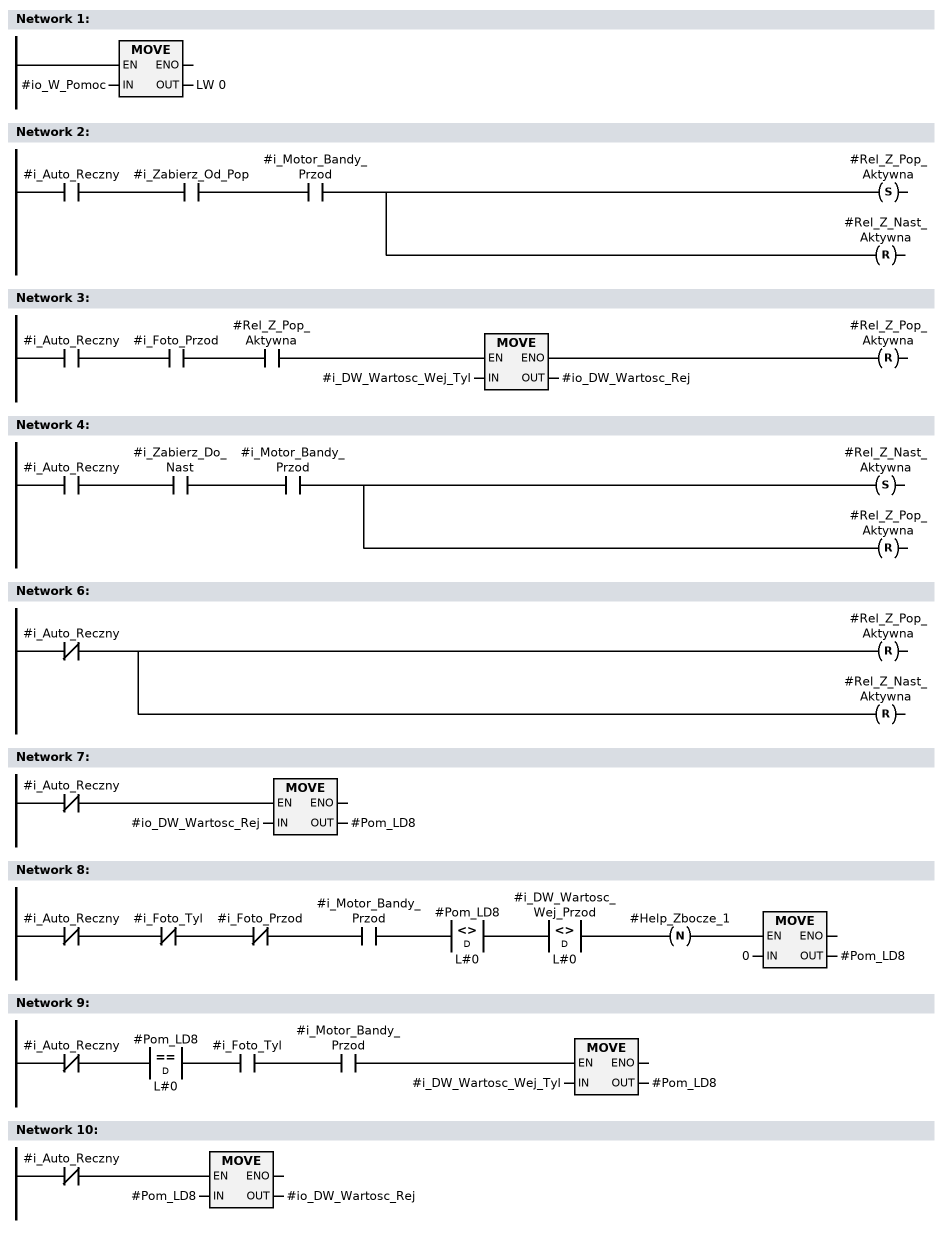
[picture p321: Monitor_Bandy_2 networks 1-10]
NETWORK
TITLE =
//Ten network celowo jest wolny
      L     #io_W_Pomoc;
      T     LW 0;
      NOP   0;
NETWORK
TITLE =
//Tryb Auto
//Pobranie wartosci
//
      A     #i_Auto_Reczny;
      A     #i_Zabierz_Od_Pop;
      A     #i_Motor_Bandy_Przod;
      S     #Rel_Z_Pop_Aktywna;
      R     #Rel_Z_Nast_Aktywna;
NETWORK
TITLE =
//Dojazd do fotokomorki i przepisanie wartosci.Informacja moze byc tez szybciej 
//przekazana (Gender potrzebuje szybciej)
      A     #i_Auto_Reczny;
      A     #i_Foto_Przod;
      A     #Rel_Z_Pop_Aktywna;
      JNB   _001;
      L     #i_DW_Wartosc_Wej_Tyl;
      T     #io_DW_Wartosc_Rej;
      SET;
      SAVE;
      CLR;
_001: A     BR;
      R     #Rel_Z_Pop_Aktywna;
NETWORK
TITLE =
//Relacja z nastepna banda
      A     #i_Auto_Reczny;
      A     #i_Zabierz_Do_Nast;
      A     #i_Motor_Bandy_Przod;
      S     #Rel_Z_Nast_Aktywna;
      R     #Rel_Z_Pop_Aktywna;
NETWORK
TITLE =
//Tryb Reczny
//Warunkiem prawidlowego dzialania trybu reczenego jest pokrycie zawsze co 
//najmniej jednej fotokomorki gdy jest produkt
//
//
NETWORK
TITLE =
//Zresetowanie relacji z automatyki
//
      AN    #i_Auto_Reczny;
      R     #Rel_Z_Pop_Aktywna;
      R     #Rel_Z_Nast_Aktywna;
NETWORK
TITLE =
//Trzeba sobie jakos radzic
      AN    #i_Auto_Reczny;
      JNB   _002;
      L     #io_DW_Wartosc_Rej;
      T     #Pom_LD8;
_002: NOP   0;
NETWORK
TITLE =
//Jazda do przodu na recznym.Bierzaca--->Nastepna
      AN    #i_Auto_Reczny;
      AN    #i_Foto_Tyl;
      AN    #i_Foto_Przod;
      A     #i_Motor_Bandy_Przod;
      A(;
      L     #Pom_LD8;
      L     L#0;
      <>D;
      );
      A(;
      L     #i_DW_Wartosc_Wej_Przod;
      L     L#0;
      <>D;
      );
      FN    #Help_Zbocze_1;
      JNB   _003;
      L     0;
      T     #Pom_LD8;
_003: NOP   0;
NETWORK
TITLE =
//Poprzednia wjezdza na bierzaca w trybie recznym. Poprzednia--->Bierzaca
      AN    #i_Auto_Reczny;
      A(;
      L     #Pom_LD8;
      L     L#0;
      ==D;
      );
      A     #i_Foto_Tyl;
      A     #i_Motor_Bandy_Przod;
      JNB   _004;
      L     #i_DW_Wartosc_Wej_Tyl;
      T     #Pom_LD8;
_004: NOP   0;
NETWORK
TITLE =
//Przepisanie powrotne
      AN    #i_Auto_Reczny;
      JNB   _005;
      L     #Pom_LD8;
      T     #io_DW_Wartosc_Rej;
_005: NOP   0;
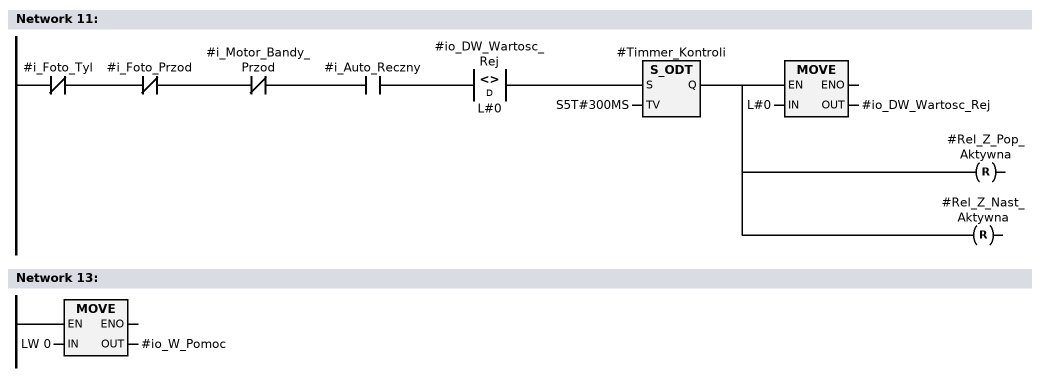
NETWORK
TITLE =
//Sprawdznie wszystkiego
//
      AN    #i_Foto_Tyl;
      AN    #i_Foto_Przod;
      AN    #i_Motor_Bandy_Przod;
      A     #i_Auto_Reczny;
      A(;
      L     #io_DW_Wartosc_Rej;
      L     L#0;
      <>D;
      );
      L     S5T#300MS;
      SD    #Timmer_Kontroli;
      NOP   0;
      NOP   0;
      NOP   0;
      A     #Timmer_Kontroli;
      =     L 12.0;
      A     L 12.0;
      JNB   _006;
      L     L#0;
      T     #io_DW_Wartosc_Rej;
_006: NOP   0;
      A     L 12.0;
      BLD   102;
      R     #Rel_Z_Pop_Aktywna;
      A     L 12.0;
      BLD   102;
      R     #Rel_Z_Nast_Aktywna;
NETWORK
TITLE =
//0.7 - paleta obecna (nieuzywane)
//0.6 - kierunek spedycja (uzywane)
//0.5 - kierunek intro (uzywane)
//0.4 - wiazanie poprzeczne (uzywane)
//0.3 - wiazanie wzdluzne   (uzywane)
//0.2 - deklowanie (uzywane)
//0.1 - foliowanie (uzywane)
//0.0 - paleta obrabiana
//1.7 - rezerwa (nieuzywane)
//1.6 - rezerwa (nieuzywane)
//1.5 - rezerwa (nieuzywane)
//1.3 - rezerwa (nieuzywane)
//1.3 - info bit 3
//1.2 - info bit 2
//1.1 - info bit 1 
//1.0 - info bit 0
//
NETWORK
TITLE =
//Przypisanie wartosci z pamieci podrecznej
//
      L     LW 0;
      T     #io_W_Pomoc;
      NOP   0;
END_FUNCTION

FUNCTION "Monitor_Palety" : VOID	// FC 316
VERSION : 0.1
VAR_INPUT
  Foto_Pozycji_Przod : BOOL ;
  Foto_Pozycji_Tyl : BOOL ;	//Opcjonalna fotokomorka
END_VAR
VAR_IN_OUT
  iod_Wartosc_Rejestru : DINT ;
END_VAR
VAR_TEMP
  Wartosc_Pomocnicz_0 : DINT ;
  Wartosc_Pomocnicz_1 : DINT ;
END_VAR
BEGIN
NETWORK
TITLE =
      L     #iod_Wartosc_Rejestru;
      T     #Wartosc_Pomocnicz_0;
      O     #Foto_Pozycji_Przod;
      O     #Foto_Pozycji_Tyl;
      JCN   et_1;
      SET;
      S     L 0.7;
et_1: NOP   0;
      AN    #Foto_Pozycji_Przod;
      AN    #Foto_Pozycji_Tyl;
      JCN   et_2;
      SET;
      R     L 0.7;
et_2: NOP   0;
      L     #Wartosc_Pomocnicz_0;
      T     #iod_Wartosc_Rejestru;
END_FUNCTION

FUNCTION "Znajdz_Widmo" : VOID	// FC 317
//0.7 - paleta obecna (nieuzywane)
//0.6 - kierunek spedycja (uzywane)
//0.5 - kierunek intro (uzywane)
//0.4 - wiazanie poprzeczne (uzywane)
//0.3 - wiazanie wzdluzne   (uzywane)
//0.2 - deklowanie (uzywane)
//0.1 - foliowanie (uzywane)
//0.0 - paleta obrabiana
//1.7 - rezerwa (nieuzywane)
//1.6 - rezerwa (nieuzywane)
//1.5 - rezerwa (nieuzywane)
//1.3 - rezerwa (nieuzywane)
//1.3 - info bit 3
//1.2 - info bit 2
//1.1 - info bit 1 
//1.0 - info bit 0
VERSION : 0.1
VAR_INPUT
  Paleta_Obecna : BOOL ;
END_VAR
VAR_IN_OUT
  iod_Wartosc_Rejestru : DINT ;
END_VAR
VAR_TEMP
  Wartosc_Pomocnicz_0 : DINT ;
  Wartosc_Pomocnicz_1 : DINT ;
END_VAR
BEGIN
NETWORK
TITLE =
      L     #iod_Wartosc_Rejestru;
      T     #Wartosc_Pomocnicz_0;
      A     #Paleta_Obecna;
      JCN   et_1;
//jesli nie wiadomo co zrobic z paleta i skad 
//jes
      AN    L 0.6;
      AN    L 0.5;
      S     L 0.5;
et_1: NOP   0;
      L     #Wartosc_Pomocnicz_0;
      T     #iod_Wartosc_Rejestru;
END_FUNCTION

FUNCTION "Dekoduj_Maske" : VOID	// FC 320
//0.0 - paleta obecna (nieuzywane)
//0.1 - kierunek spedycja (uzywane)
//0.2 - kierunek intro (uzywane)
//0.3 - wiazanie poprzeczne (uzywane)
//0.4 - wiazanie wzdluzne   (uzywane)
//0.5 - deklowanie (uzywane)
//0.6 - foliowanie (uzywane)
//0.7 - paleta_obrabiana
//1.0 - info bit 0
//1.1 - info bit 1
//1.2 - info bit 2 
//1.3 - info bit 3
//1.4 - rezerwa (nieuzywane)
//1.5 - rezerwa (nieuzywane)
//1.6 - rezerwa (nieuzywane)
//1.7 - rezerwa (nieuzywane)
//
VERSION : 0.1
VAR_INPUT
  Wartosc_Elementu : DINT ;
END_VAR
VAR_OUTPUT
  o_Paleta_Obecna : BOOL ;	//0.7
  o_Kierunek_Spedycja : BOOL ;	//0.6
  o_Kierunek_Intro : BOOL ;	//0.5
  o_Wizanie_Poprzeczne : BOOL ;	//0.4
  o_Wiazanie_Wzdluzne : BOOL ;	//0.3
  o_Deklowanie : BOOL ;	//0.2
  o_Foliowanie : BOOL ;	//0.1
  o_Paleta_Obrabiana : BOOL ;	//0.0
  o_Rezerwa_1_7 : BOOL ;	//1.7
  o_Rezerwa_1_6 : BOOL ;	//1.1
  o_Rezerwa_1_5 : BOOL ;	//1.2
  o_Rezerwa_1_4 : BOOL ;	//1.4
  o_Info_Bit_3 : BOOL ;	//1.3
  o_Info_Bit_2 : BOOL ;	//1.2
  o_Info_Bit_1 : BOOL ;	//1.1
  o_Info_Bit_0 : BOOL ;	//1.0
END_VAR
VAR_TEMP
  Edek_0 : DWORD ;
  Paleta_Obrabiana : BOOL ;	//0.0 - paleta_obrabiana
  Foliowanie : BOOL ;	//0.1
  Deklowanie : BOOL ;	//0.2
  Wiazanie_Wzdluzne : BOOL ;	//0.3
  Wizanie_Poprzeczne : BOOL ;	//0.4
  Kierunek_Intro : BOOL ;	//0.5
  Kierunek_Spedycja : BOOL ;	//0.6
  Paleta_Obecna : BOOL ;	//0.7
  Info_Bit_0 : BOOL ;	//1.0
  Info_Bit_1 : BOOL ;	//1.1
  Info_Bit_2 : BOOL ;	//1.2
  Info_Bit_3 : BOOL ;	//1.3
  Rezerwa_1_4 : BOOL ;	//1.4
  Rezerwa_1_5 : BOOL ;	//1.5
  Rezerwa_1_6 : BOOL ;	//1.6
  Rezerwa_1_7 : BOOL ;	//1.7
END_VAR
BEGIN
NETWORK
TITLE =
//ten network celowo jest wolny
NETWORK
TITLE =
//Zaladowanie maski
      L     #Wartosc_Elementu;
      T     LD 4;
NETWORK
TITLE =
//Wyluskanie zadan
      A     #Paleta_Obrabiana;
      =     #o_Paleta_Obrabiana;
//***
      A     #Foliowanie;
      =     #o_Foliowanie;
//***
      A     #Deklowanie;
      =     #o_Deklowanie;
//***
      A     #Wiazanie_Wzdluzne;
      =     #o_Wiazanie_Wzdluzne;
//***
      A     #Wizanie_Poprzeczne;
      =     #o_Wizanie_Poprzeczne;
//***
      A     #Kierunek_Intro;
      =     #o_Kierunek_Intro;
//***
      A     #Kierunek_Spedycja;
      =     #o_Kierunek_Spedycja;
//***
      A     #Paleta_Obecna;
      =     #o_Paleta_Obecna;
//***
      A     #Info_Bit_0;
      =     #o_Info_Bit_0;
//***
      A     #Info_Bit_1;
      =     #o_Info_Bit_1;
//***
      A     #Info_Bit_2;
      =     #o_Info_Bit_2;
//***
      A     #Info_Bit_3;
      =     #o_Info_Bit_3;
//***
      A     #Rezerwa_1_4;
      =     #o_Rezerwa_1_4;
//***
      A     #Rezerwa_1_5;
      =     #o_Rezerwa_1_5;
//***
      A     #Rezerwa_1_6;
      =     #o_Rezerwa_1_6;
//***
      A     #Rezerwa_1_7;
      =     #o_Rezerwa_1_7;
END_FUNCTION

FUNCTION "Dobor_Elementow_Lini" : VOID	// FC 400
//Funkcja tworzy liste przyciskow bistabilny uzywanych do wyboru trybu pracy w 
//Gender Fedder Line.Dostepne funkcjonalosci wybieramy za pomoca przyciskow
//Spedycja i Intro. Po wyborze przycisku rozwijaja sie funkcjonalnosci.
//
//Spedycja   lub  Intro:
//Spedycja->o_Wiazanie_Pop_Aktywne->o_Deklowanie_Aktywne
//Spedycja->o_Wiazanie_Wzdl_Aktywne
//Spedycja->o_Foliowanie_Aktywne
//
//Intro->o_Instert_Intro_Aktywne
//
//Na koncu funkcji tworzona jest mask sluzaca dalszej obrobce zadan w programie.
//Bity maski:
//
//0.7 - paleta obecna (nieuzywane)
//0.6 - kierunek spedycja (uzywane)
//0.5 - kierunek intro (uzywane)
//0.4 - wiazanie poprzeczne (uzywane)
//0.3 - wiazanie wzdluzne   (uzywane)
//0.2 - deklowanie (uzywane)
//0.1 - foliowanie (uzywane)
//0.0 - paleta obrabiana
//1.7 - rezerwa (nieuzywane)
//1.6 - rezerwa (nieuzywane)
//1.5 - rezerwa (nieuzywane)
//1.3 - rezerwa (nieuzywane)
//1.3 - info bit 3
//1.2 - info bit 2
//1.1 - info bit 1 
//1.0 - info bit 0
//
AUTHOR : Kng
NAME : Help_FC
VERSION : 0.1
VAR_INPUT
  i_Kierunek_Spedycja : BOOL ;
  i_Kierunek_Intro : BOOL ;
  i_Wiazanie_Poprzeczne : BOOL ;
  i_Wiazanie_Wzdluzne : BOOL ;
  i_Deklowanie : BOOL ;
  i_Foliowanie : BOOL ;
  i_Paleta_Obrabiana : BOOL ;	//Informacja czy paleta jest obrabiana
  i_Koder_Bit_0 : BOOL ;
  i_Koder_Bit_1 : BOOL ;
  i_Koder_Bit_2 : BOOL ;
  i_Koder_Bit_3 : BOOL ;
END_VAR
VAR_OUTPUT
  o_Kier_Spedycja_Wyb : BOOL ;
  o_Kier_Intro_Wyb : BOOL ;
  o_Wiazanie_Pop_Wyb : BOOL ;	//To co jest wybrane
  o_Wiazanie_Wzdl_Wyb : BOOL ;
  o_Deklowanie_Wyb : BOOL ;
  o_Foliowanie_Wyb : BOOL ;
  o_Kier_Spedycja_Akt : BOOL ;
  o_Kier_Intro_Akt : BOOL ;
  o_Wiazanie_Pop_Akt : BOOL ;	//To co mozna wybrac
  o_Wiazanie_Wzdl_Akt : BOOL ;
  o_Deklowanie_Akt : BOOL ;
  o_Foliowanie_Akt : BOOL ;
  o_Maska_Zadania : INT ;	//Maska w wynikowa
END_VAR
VAR_IN_OUT
  io_Help_DW : DINT ;	//Slowo pomocnicze
END_VAR
VAR_TEMP
  L_Rezerwa_0_0 : BOOL ;
  L_Rezerwa_0_1 : BOOL ;
  L_Rezerwa_0_2 : BOOL ;
  L_Rezerwa_0_3 : BOOL ;
  L_Rezerwa_0_4 : BOOL ;
  L_Rezerwa_0_5 : BOOL ;
  L_Rezerwa_0_6 : BOOL ;
  L_Rezerwa_0_7 : BOOL ;
  L_Rezerwa_1_0 : BOOL ;
  L_Rezerwa_1_1 : BOOL ;
  L_Rezerwa_1_2 : BOOL ;
  L_Rezerwa_1_3 : BOOL ;
  L_Rezerwa_1_4 : BOOL ;
  L_Rezerwa_1_5 : BOOL ;
  L_Rezerwa_1_6 : BOOL ;
  L_Rezerwa_1_7 : BOOL ;
  L_Rezerwa_Int_2_0 : INT ;
  io_L_Kier_Spedycja : BOOL ;
  io_L_Wiazanie_Poprzeczne : BOOL ;
  io_L_Wiazanie_Wzdluzne : BOOL ;
  io_L_Deklowanie : BOOL ;
  io_L_Foliowanie : BOOL ;
  io_L_Kier_Insert_Intro : BOOL ;
  io_L_Help_Bit_0 : BOOL ;
  io_L_Help_Bit_1 : BOOL ;
  io_L_Help_Bit_2 : BOOL ;
  io_L_Help_Bit_3 : BOOL ;
  io_L_Help_Bit_4 : BOOL ;
  io_L_Help_Bit_5 : BOOL ;
  io_L_Help_Bit_6 : BOOL ;
  L_Rezerwa_Int_6_0 : INT ;
  L_Paleta_Obrabiana : BOOL ;
  L_Foliowanie : BOOL ;
  L_Deklowanie : BOOL ;
  L_Wiazanie_Wzdluzne : BOOL ;
  L_Wiazanie_Poprzeczne : BOOL ;
  L_Kierunek_Intro : BOOL ;
  L_Kierunek_Spedycja : BOOL ;
  L_Paleta_Obecna : BOOL ;
  L_Info_Bit_0 : BOOL ;
  L_Info_Bit_1 : BOOL ;
  L_Info_Bit_2 : BOOL ;
  L_Info_Bit_3 : BOOL ;
  L_Rezerwa_9_4 : BOOL ;
  L_Rezerwa_9_5 : BOOL ;
  L_Rezerwa_9_6 : BOOL ;
  L_Rezerwa_9_7 : BOOL ;
END_VAR
BEGIN
NETWORK
TITLE =
//Ten network celowo jest wolny
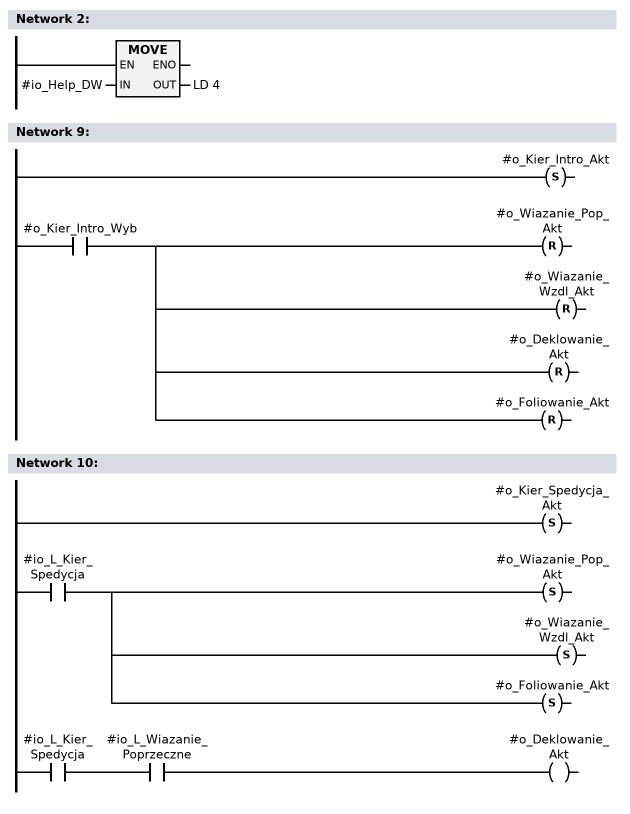
NETWORK
TITLE =
      L     #io_Help_DW;
      T     LD 4;
NETWORK
TITLE =
//Spedycja lub intro
      A(;
      A     #i_Kierunek_Spedycja;
      FP    #io_L_Help_Bit_5;
      S     #io_L_Kier_Spedycja;
      A     #i_Kierunek_Intro;
      FP    #io_L_Help_Bit_4;
      R     #io_L_Kier_Spedycja;
      A     #io_L_Kier_Spedycja;
      );
      NOT;
      =     #io_L_Kier_Insert_Intro;
NETWORK
TITLE =
//Wiazanie poprzeczne
// (network holds code this reader does not know; not shown)
NETWORK
TITLE =
//Wiazanie Wzdluzne
// (network holds code this reader does not know; not shown)
NETWORK
TITLE =
//Deklowanie
// (network holds code this reader does not know; not shown)
NETWORK
TITLE =
//Foliowanie
// (network holds code this reader does not know; not shown)
NETWORK
TITLE =
NETWORK
TITLE =
//Kierunek Insert
//Kierunek intro zawsze mozliwy do wyboru
      SET;
      S     #o_Kier_Intro_Akt;
      A     #o_Kier_Intro_Wyb;
      R     #o_Wiazanie_Pop_Akt;
      R     #o_Wiazanie_Wzdl_Akt;
      R     #o_Deklowanie_Akt;
      R     #o_Foliowanie_Akt;
NETWORK
TITLE =
//Kierunek spedycja
//
//Kierunek spedycja zawsze mozliwy do wyboru
      SET;
      S     #o_Kier_Spedycja_Akt;
      A     #io_L_Kier_Spedycja;
      S     #o_Wiazanie_Pop_Akt;
      S     #o_Wiazanie_Wzdl_Akt;
      S     #o_Foliowanie_Akt;
//Wyjatek dla deklowania
      A     #io_L_Kier_Spedycja;
      A     #io_L_Wiazanie_Poprzeczne;
      =     #o_Deklowanie_Akt;
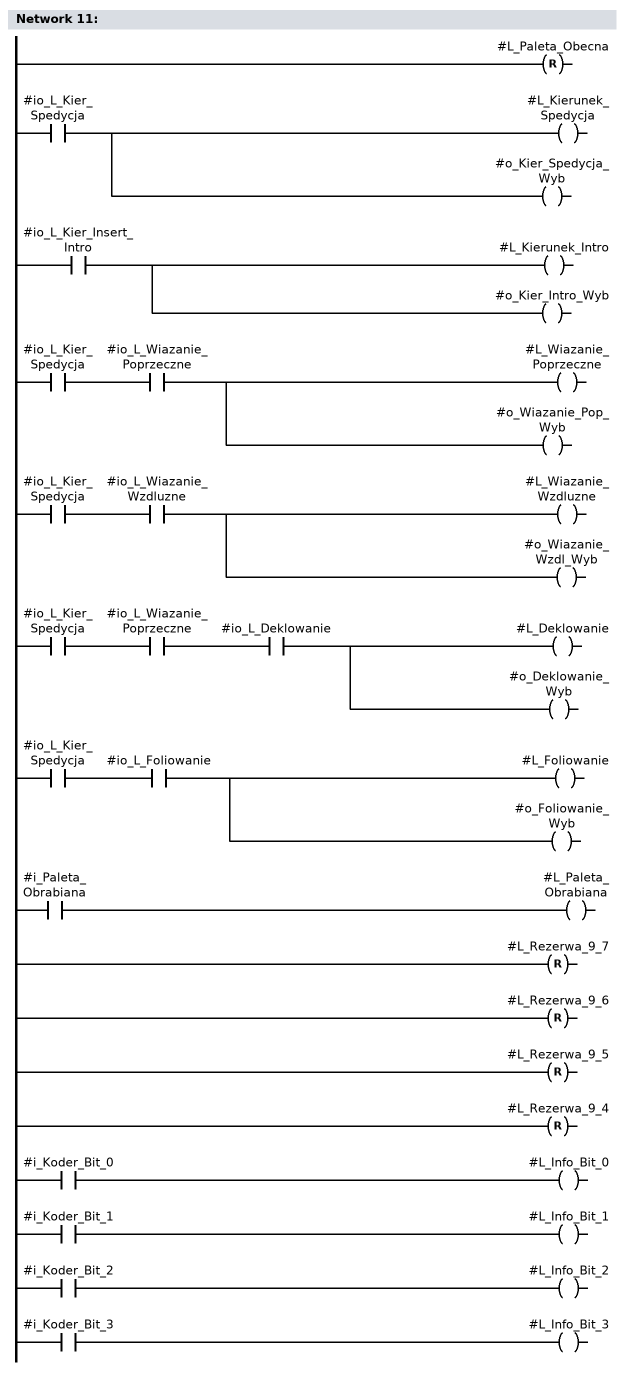
NETWORK
TITLE =
//Zakladanie maski
//0.7 - paleta obecna (nieuzywane)
//0.6 - kierunek spedycja (uzywane)
//0.5 - kierunek intro (uzywane)
//0.4 - wiazanie poprzeczne (uzywane)
//0.3 - wiazanie wzdluzne   (uzywane)
//0.2 - deklowanie (uzywane)
//0.1 - foliowanie (uzywane)
//0.0 - paleta obrabiana
//1.7 - rezerwa (nieuzywane)
//1.6 - rezerwa (nieuzywane)
//1.5 - rezerwa (nieuzywane)
//1.3 - rezerwa (nieuzywane)
//1.3 - info bit 3
//1.2 - info bit 2
//1.1 - info bit 1 
//1.0 - info bit 0
//
////Funckja sprawdzona w plcsim 
//
//***0.7 - paleta obecna (nieuzywane)
      SET;
      R     #L_Paleta_Obecna;
//***0.6 - kierunek spedycja (uzywane)
      A     #io_L_Kier_Spedycja;
      =     #L_Kierunek_Spedycja;
      =     #o_Kier_Spedycja_Wyb;
//*** 0.5 - kierunek intro (uzywane)
      A     #io_L_Kier_Insert_Intro;
      =     #L_Kierunek_Intro;
      =     #o_Kier_Intro_Wyb;
//*** 0.4 - wiazanie poprzeczne (uzywane)
      A     #io_L_Kier_Spedycja;
      A     #io_L_Wiazanie_Poprzeczne;
      =     #L_Wiazanie_Poprzeczne;
      =     #o_Wiazanie_Pop_Wyb;
//*** 0.3 - wiazanie wzdluzne   (uzywane)
      A     #io_L_Kier_Spedycja;
      A     #io_L_Wiazanie_Wzdluzne;
      =     #L_Wiazanie_Wzdluzne;
      =     #o_Wiazanie_Wzdl_Wyb;
//*** 0.2 - deklowanie (uzywane)
      A     #io_L_Kier_Spedycja;
      A     #io_L_Wiazanie_Poprzeczne;
      A     #io_L_Deklowanie;
      =     #L_Deklowanie;
      =     #o_Deklowanie_Wyb;
//*** 0.1 - foliowanie (uzywane)
      A     #io_L_Kier_Spedycja;
      A     #io_L_Foliowanie;
      =     #L_Foliowanie;
      =     #o_Foliowanie_Wyb;
//*** 1.0 - info paleta obrabiana
      A     #i_Paleta_Obrabiana;
      =     #L_Paleta_Obrabiana;
//*** 1.7 - rezerwa (nieuzywane)
      SET;
      R     #L_Rezerwa_9_7;
//*** 1.6 - rezerwa (nieuzywane)
      SET;
      R     #L_Rezerwa_9_6;
//*** 1.5 - rezerwa (nieuzywane)
      SET;
      R     #L_Rezerwa_9_5;
//*** 1.4 - rezerwa (nieuzywane)
      SET;
      R     #L_Rezerwa_9_4;
//*** 1.3 - info bit 0
      A     #i_Koder_Bit_0;
      =     #L_Info_Bit_0;
//*** 1.2 - info bit 1
      A     #i_Koder_Bit_1;
      =     #L_Info_Bit_1;
//*** 1.1 - info bit 2 
      A     #i_Koder_Bit_2;
      =     #L_Info_Bit_2;
//*** 1.0 - info bit 3
      A     #i_Koder_Bit_3;
      =     #L_Info_Bit_3;
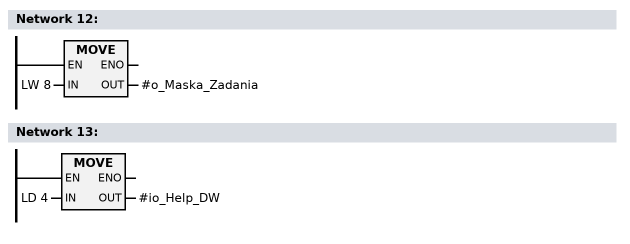
NETWORK
TITLE =
//Przypisz maske
      L     LW 8;
      T     #o_Maska_Zadania;
NETWORK
TITLE =
//Przypisz bity przejsciowe
      L     LD 4;
      T     #io_Help_DW;
END_FUNCTION

FUNCTION "Wozek_Queue_V3" : VOID	// FC 408
AUTHOR : Kng
NAME : Fahren
VERSION : 0.1
VAR_INPUT
  _Paleta_KB1 : BOOL ;
  Kier_KB1_Gender : BOOL ;
  Kier_KB1_Intro : BOOL ;
  Wartosc_KB1 : INT ;
  Kod_KB1 : BYTE ;
  _Paleta_KB2 : BOOL ;
  Kier_KB2_Gender : BOOL ;
  Kier_KB2_Intro : BOOL ;
  Wartosc_KB2 : INT ;
  Kod_KB2 : BYTE ;
  _Paleta_I1 : BOOL ;	//Intro pobieranie nr 1
  Kier_I1_Gender : BOOL ;
  Kier_I1_Intro : BOOL ;
  Wartosc_I1 : INT ;
  Kod_I1 : BYTE ;
  _Paleta_I2 : BOOL ;	//Intro pobieranie nr 2
  Kier_I2_Gender : BOOL ;
  Kier_I2_Intro : BOOL ;
  Wartosc_I2 : INT ;
  Kod_I2 : BYTE ;
  _Paleta_I3 : BOOL ;	//Intro pobieranie nr 2
  Kier_I3_Gender : BOOL ;
  Kier_I3_Intro : BOOL ;
  Wartosc_I3 : INT ;
  Kod_I3 : BYTE ;
END_VAR
VAR_OUTPUT
  od_Wartosc_KB1 : DINT ;
  od_Wartosc_KB2 : DINT ;
  od_Wartosc_I1 : DINT ;
  od_Wartosc_I2 : DINT ;
  od_Wartosc_I3 : DINT ;
END_VAR
VAR_TEMP
  Slowo_LW0 : INT ;
  Slowo_LW2 : INT ;
  Temp_Help_1 : BOOL ;
END_VAR
BEGIN
NETWORK
TITLE =
//Ten Network celowo jest wolny
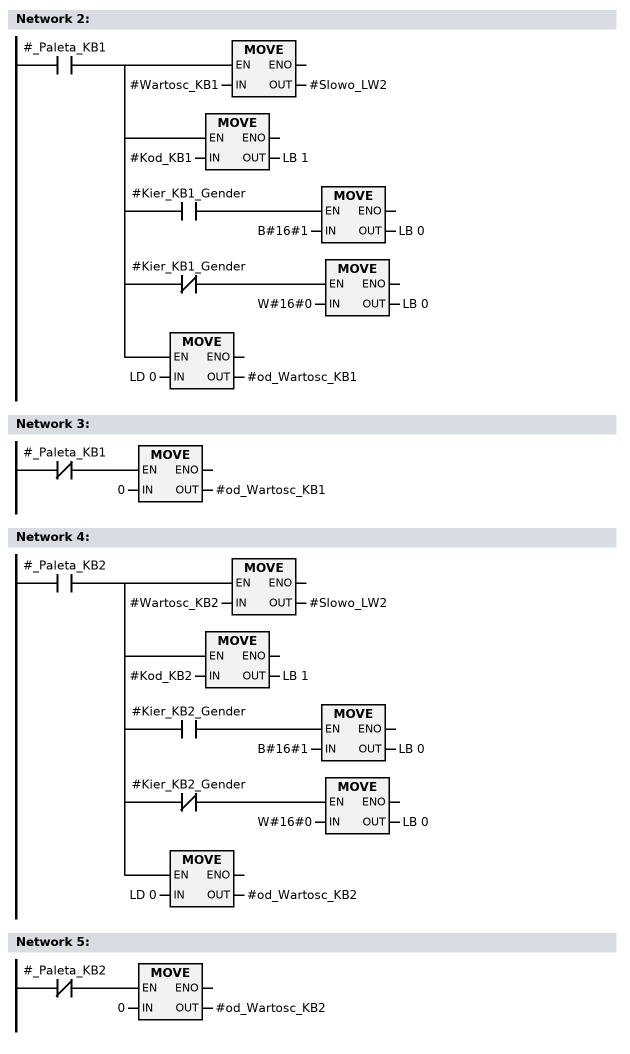
NETWORK
TITLE =
//Budowanie wartosci transferowej :
//LB0-kierunek intro(1),spedycja(0)
//LB1-Kod maszyny np KB1-1
//LW2-Wartosc wagowa
      A     #_Paleta_KB1;
      =     L 5.0;
      A     L 5.0;
      JNB   _001;
      L     #Wartosc_KB1;
      T     #Slowo_LW2;
_001: NOP   0;
      A     L 5.0;
      JNB   _002;
      L     #Kod_KB1;
      T     LB 1;
_002: NOP   0;
      A     L 5.0;
      A     #Kier_KB1_Gender;
      JNB   _003;
      L     B#16#1;
      T     LB 0;
_003: NOP   0;
      A     L 5.0;
      AN    #Kier_KB1_Gender;
      JNB   _004;
      L     W#16#0;
      T     LB 0;
_004: NOP   0;
      A     L 5.0;
      JNB   _005;
      L     LD 0;
      T     #od_Wartosc_KB1;
_005: NOP   0;
NETWORK
TITLE =
      AN    #_Paleta_KB1;
      JNB   _006;
      L     0;
      T     #od_Wartosc_KB1;
_006: NOP   0;
NETWORK
TITLE =
//Budowanie wartosci transferowej dla kb2
      A     #_Paleta_KB2;
      =     L 5.0;
      A     L 5.0;
      JNB   _007;
      L     #Wartosc_KB2;
      T     #Slowo_LW2;
_007: NOP   0;
      A     L 5.0;
      JNB   _008;
      L     #Kod_KB2;
      T     LB 1;
_008: NOP   0;
      A     L 5.0;
      A     #Kier_KB2_Gender;
      JNB   _009;
      L     B#16#1;
      T     LB 0;
_009: NOP   0;
      A     L 5.0;
      AN    #Kier_KB2_Gender;
      JNB   _00a;
      L     W#16#0;
      T     LB 0;
_00a: NOP   0;
      A     L 5.0;
      JNB   _00b;
      L     LD 0;
      T     #od_Wartosc_KB2;
_00b: NOP   0;
NETWORK
TITLE =
//jezeli brak palety na kb2 to przypisz 0
      AN    #_Paleta_KB2;
      JNB   _00c;
      L     0;
      T     #od_Wartosc_KB2;
_00c: NOP   0;
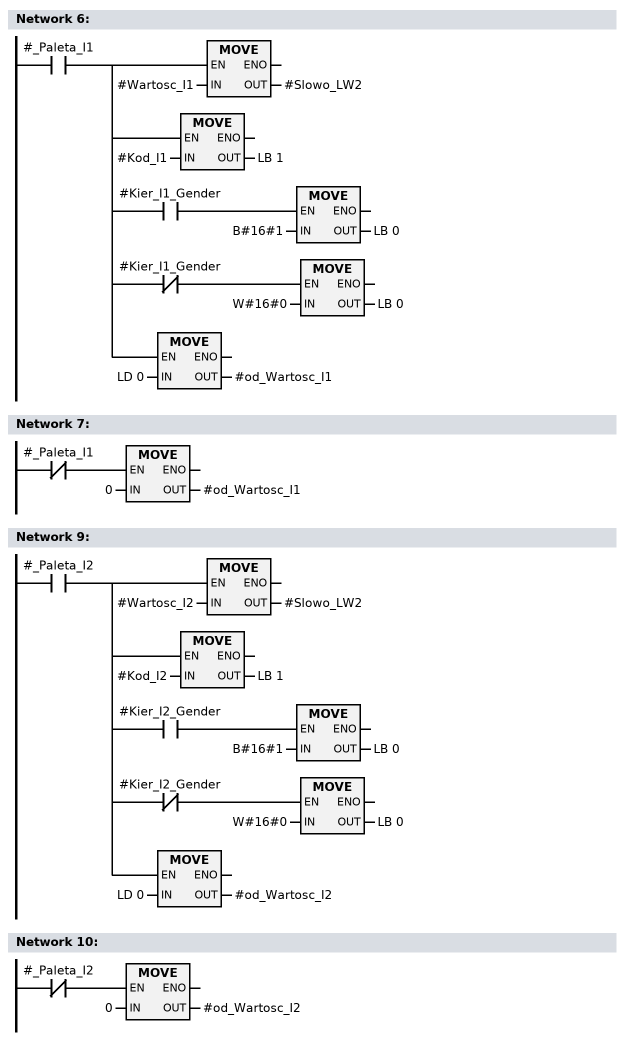
NETWORK
TITLE =
//Budowanie wartosci transferowej dla intro
      A     #_Paleta_I1;
      =     L 5.0;
      A     L 5.0;
      JNB   _00d;
      L     #Wartosc_I1;
      T     #Slowo_LW2;
_00d: NOP   0;
      A     L 5.0;
      JNB   _00e;
      L     #Kod_I1;
      T     LB 1;
_00e: NOP   0;
      A     L 5.0;
      A     #Kier_I1_Gender;
      JNB   _00f;
      L     B#16#1;
      T     LB 0;
_00f: NOP   0;
      A     L 5.0;
      AN    #Kier_I1_Gender;
      JNB   _010;
      L     W#16#0;
      T     LB 0;
_010: NOP   0;
      A     L 5.0;
      JNB   _011;
      L     LD 0;
      T     #od_Wartosc_I1;
_011: NOP   0;
NETWORK
TITLE =
      AN    #_Paleta_I1;
      JNB   _012;
      L     0;
      T     #od_Wartosc_I1;
_012: NOP   0;
NETWORK
TITLE =
NETWORK
TITLE =
//Budowanie wartosci transferowej dla intro
      A     #_Paleta_I2;
      =     L 5.0;
      A     L 5.0;
      JNB   _013;
      L     #Wartosc_I2;
      T     #Slowo_LW2;
_013: NOP   0;
      A     L 5.0;
      JNB   _014;
      L     #Kod_I2;
      T     LB 1;
_014: NOP   0;
      A     L 5.0;
      A     #Kier_I2_Gender;
      JNB   _015;
      L     B#16#1;
      T     LB 0;
_015: NOP   0;
      A     L 5.0;
      AN    #Kier_I2_Gender;
      JNB   _016;
      L     W#16#0;
      T     LB 0;
_016: NOP   0;
      A     L 5.0;
      JNB   _017;
      L     LD 0;
      T     #od_Wartosc_I2;
_017: NOP   0;
NETWORK
TITLE =
//Kasuj buffor dla I2
      AN    #_Paleta_I2;
      JNB   _018;
      L     0;
      T     #od_Wartosc_I2;
_018: NOP   0;
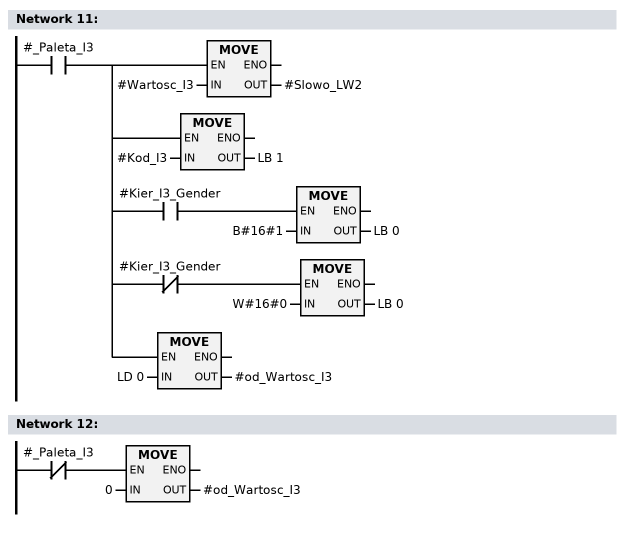
NETWORK
TITLE =
//Budowanie wartosci transferowej dla intro
      A     #_Paleta_I3;
      =     L 5.0;
      A     L 5.0;
      JNB   _019;
      L     #Wartosc_I3;
      T     #Slowo_LW2;
_019: NOP   0;
      A     L 5.0;
      JNB   _01a;
      L     #Kod_I3;
      T     LB 1;
_01a: NOP   0;
      A     L 5.0;
      A     #Kier_I3_Gender;
      JNB   _01b;
      L     B#16#1;
      T     LB 0;
_01b: NOP   0;
      A     L 5.0;
      AN    #Kier_I3_Gender;
      JNB   _01c;
      L     W#16#0;
      T     LB 0;
_01c: NOP   0;
      A     L 5.0;
      JNB   _01d;
      L     LD 0;
      T     #od_Wartosc_I3;
_01d: NOP   0;
NETWORK
TITLE =
//Kasuj buffor dla I2
      AN    #_Paleta_I3;
      JNB   _01e;
      L     0;
      T     #od_Wartosc_I3;
_01e: NOP   0;
END_FUNCTION

FUNCTION "Sorting_V3" : VOID	// FC 409
//Funkcja odpowiada za sortowanie elementow dostarczonych do bloku db. Sortowanie 
//odbywa sie automatcycznie. Wpisanie nastepuje przez zbocze na wejsciu wpisz 
//wartosc.
//
//Funkcja odnosi sie bezposrednio do bloku danych db402
//
//
//
//
AUTHOR : Kng
NAME : Help_FC
VERSION : 0.1
VAR_INPUT
  id_Wartosc_KB1 : DINT ;	//Wpisuje nowy rekord na dol bloku
  id_Wartosc_KB2 : DINT ;	//Pobiera rekord z gory bloku
  id_Wartosc_I1 : DINT ;	//Kasuje rekord od wartosci wsadowej
  id_Wartosc_I2 : DINT ;
  id_Wartosc_I3 : DINT ;
  i_Poz_5_Down : BOOL ;
  i_Poz_4_Up : BOOL ;
  i_Poz_4_Down : BOOL ;
  i_Poz_3_Up : BOOL ;
  i_Poz_3_Down : BOOL ;
  i_Poz_2_Up : BOOL ;
  i_Poz_2_Down : BOOL ;
  i_Poz_1_Up : BOOL ;
END_VAR
VAR_IN_OUT
  iow_Help_DWord : DWORD ;
END_VAR
VAR_TEMP
  P : STRUCT
   KB1_Wpis : BOOL ;
   KB2_Wpis : BOOL ;
   I1_Wpis : BOOL ;
   I2_Wpis : BOOL ;
   I3_Wpis : BOOL ;
   KB1_Istnieje : BOOL ;
   KB2_Istnieje : BOOL ;
   I1_Istnieje : BOOL ;
   I2_Istnieje : BOOL ;
   I3_Istnieje : BOOL ;
   Help_Bit_0_7 : BOOL ;
   Wpis_0_istnieje : BOOL ;
   Wpis_1_istnieje : BOOL ;
   Wpis_2_istnieje : BOOL ;
   Wpis_3_istnieje : BOOL ;
   Wpis_4_istnieje : BOOL ;
   Wpis_5_istnieje : BOOL ;
   Wpis_6_istnieje : BOOL ;
   edge_1 : BOOL ;
   edge_2 : BOOL ;
   edge_3 : BOOL ;
   edge_4 : BOOL ;
   edge_5 : BOOL ;
   edge_6 : BOOL ;
  END_STRUCT ;
  Help_Blok_Move : INT ;
  Help_Int_2 : INT ;
  Help_Dint : DINT ;
  Wpis : STRUCT
   _0_dbb0_Kod_Kier : BYTE ;
   _0_dbb1_Kod_Maszyna : BYTE ;
   _0_dbw2_War_Wagowa : INT ;
   _1_dbb4_Kod_Kier : BYTE ;
   _1_dbb5_Kod_Maszyna : BYTE ;
   _1_dbw6_War_Wagowa : INT ;
   _2_dbb8_Kod_Kier : BYTE ;
   _2_dbb9_Kod_Maszyna : BYTE ;
   _2_dbw10_War_Wagowa : INT ;
   _3_dbb12_Kod_Kier : BYTE ;
   _3_dbb13_Kod_Maszyna : BYTE ;
   _3_dbw14_War_Wagowa : INT ;
   _4_dbb16_Kod_Kier : BYTE ;
   _4_dbb17_Kod_Maszyna : BYTE ;
   _4_dbw18_War_Wagowa : INT ;
   _5_dbb20_Kod_Kier : BYTE ;
   _5_dbb21_Kod_Masz : BYTE ;
   _5_dbw22_War_Wagowa : INT ;
   _6_dbb24_Kod_Kier : BYTE ;
   _6_dbb25_Kod_Masz : BYTE ;
   _6_dbw26_War_Wagowa : INT ;
   Kod_Spr_KB1 : BYTE ;
   Kod_Spr_KB2 : BYTE ;
   Kod_Spr_I1 : BYTE ;
   Kod_Spr_I2 : BYTE ;
   Kod_Spr_I3 : BYTE ;
   Kod_Spr_Rezerwa : BYTE ;
  END_STRUCT ;
  Temp_Wpis_KB1 : BOOL ;
  Temp_Wpis_KB2 : BOOL ;
  Temp_Wpis_I1 : BOOL ;
  Temp_Wpis_I2 : BOOL ;
  Temp_Wpis_I3 : BOOL ;
END_VAR
BEGIN
NETWORK
TITLE =
//Ten Network celowo jest wolny
NETWORK
TITLE =
//Zaladowanie bitow przejsciowych
      L     #iow_Help_DWord;
      T     #P;
//Zaladowanie pakietu danych
      CALL  "BLKMOV" (
           SRCBLK                   := "Key_DB".Wpis,
           RET_VAL                  := #Help_Blok_Move,
           DSTBLK                   := #Wpis);
NETWORK
TITLE =
//Sprawdz istniejacy wpis
      L     #id_Wartosc_KB1;
      L     0;
      <>D;
      =     #P.KB1_Istnieje;
      NOT;
      R     #P.KB1_Wpis;
//---
      L     #id_Wartosc_KB2;
      L     0;
      <>D;
      =     #P.KB2_Istnieje;
      NOT;
      R     #P.KB2_Wpis;
//---
      L     #id_Wartosc_I1;
      L     0;
      <>D;
      =     #P.I1_Istnieje;
      NOT;
      R     #P.I1_Wpis;
//---
      L     #id_Wartosc_I2;
      L     0;
      <>D;
      =     #P.I2_Istnieje;
      NOT;
      R     #P.I2_Wpis;
//---
      L     #id_Wartosc_I3;
      L     0;
      <>D;
      =     #P.I3_Istnieje;
      NOT;
      R     #P.I3_Wpis;
NETWORK
TITLE =
//Zaladuj kody maszyn do sprawdzenia
//****KB1*************************************
      L     #id_Wartosc_KB1;
      T     #Help_Dint;
//Zaladuj bit odpowiedzialny za maszyne (kod maszyny)
      L     LB 9;
      T     #Wpis.Kod_Spr_KB1;
//****KB2*************************************
      L     #id_Wartosc_KB2;
      T     #Help_Dint;
//Zaladuj bit odpowiedzialny za maszyne (kod maszyny)
      L     LB 9;
      T     #Wpis.Kod_Spr_KB2;
//****I1**************************************
      L     #id_Wartosc_I1;
      T     #Help_Dint;
//Zaladuj bit odpowiedzialny za maszyne (kod maszyny)
      L     LB 9;
      T     #Wpis.Kod_Spr_I1;
//****I2**************************************
      L     #id_Wartosc_I2;
      T     #Help_Dint;
//Zaladuj bit odpowiedzialny za maszyne (kod maszyny)
      L     LB 9;
      T     #Wpis.Kod_Spr_I2;
//****I3**************************************
      L     #id_Wartosc_I3;
      T     #Help_Dint;
//Zaladuj bit odpowiedzialny za maszyne (kod maszyny)
      L     LB 9;
      T     #Wpis.Kod_Spr_I3;
//Przeprowadzeni sprwdzenia   dbd 0
      O(;
      L     #Wpis._0_dbb1_Kod_Maszyna;
      L     #Wpis.Kod_Spr_KB1;
      ==I;
      );
      O(;
      L     #Wpis._0_dbb1_Kod_Maszyna;
      L     #Wpis.Kod_Spr_KB2;
      ==I;
      );
      O(;
      L     #Wpis._0_dbb1_Kod_Maszyna;
      L     #Wpis.Kod_Spr_I1;
      ==I;
      );
      O(;
      L     #Wpis._0_dbb1_Kod_Maszyna;
      L     #Wpis.Kod_Spr_I2;
      ==I;
      );
      O(;
      L     #Wpis._0_dbb1_Kod_Maszyna;
      L     #Wpis.Kod_Spr_I3;
      ==I;
      );
      JC    dbd0;
      L     0;
      T     #Wpis._0_dbb0_Kod_Kier;
      T     #Wpis._0_dbb1_Kod_Maszyna;
      T     #Wpis._0_dbw2_War_Wagowa;
dbd0: NOP   0;
//Przeprowadzeni sprwdzenia   dbd 4 (pozycja 2)
      O(;
      L     #Wpis._1_dbb5_Kod_Maszyna;
      L     #Wpis.Kod_Spr_KB1;
      ==I;
      );
      O(;
      L     #Wpis._1_dbb5_Kod_Maszyna;
      L     #Wpis.Kod_Spr_KB2;
      ==I;
      );
      O(;
      L     #Wpis._1_dbb5_Kod_Maszyna;
      L     #Wpis.Kod_Spr_I1;
      ==I;
      );
      O(;
      L     #Wpis._1_dbb5_Kod_Maszyna;
      L     #Wpis.Kod_Spr_I2;
      ==I;
      );
      O(;
      L     #Wpis._1_dbb5_Kod_Maszyna;
      L     #Wpis.Kod_Spr_I3;
      ==I;
      );
      JC    dbd4;
      L     0;
      T     #Wpis._1_dbb4_Kod_Kier;
      T     #Wpis._1_dbb5_Kod_Maszyna;
      T     #Wpis._1_dbw6_War_Wagowa;
dbd4: NOP   0;
//Przeprowadzeni sprwdzenia   dbd 8 (pozycja 3)
      O(;
      L     #Wpis._2_dbb9_Kod_Maszyna;
      L     #Wpis.Kod_Spr_KB1;
      ==I;
      );
      O(;
      L     #Wpis._2_dbb9_Kod_Maszyna;
      L     #Wpis.Kod_Spr_KB2;
      ==I;
      );
      O(;
      L     #Wpis._2_dbb9_Kod_Maszyna;
      L     #Wpis.Kod_Spr_I1;
      ==I;
      );
      O(;
      L     #Wpis._2_dbb9_Kod_Maszyna;
      L     #Wpis.Kod_Spr_I2;
      ==I;
      );
      O(;
      L     #Wpis._2_dbb9_Kod_Maszyna;
      L     #Wpis.Kod_Spr_I3;
      ==I;
      );
      JC    dbd8;
      L     0;
      T     #Wpis._2_dbb8_Kod_Kier;
      T     #Wpis._2_dbb9_Kod_Maszyna;
      T     #Wpis._2_dbw10_War_Wagowa;
dbd8: NOP   0;
//Przeprowadzeni sprwdzenia   dbd 12 (pozycja 4)
      O(;
      L     #Wpis._3_dbb13_Kod_Maszyna;
      L     #Wpis.Kod_Spr_KB1;
      ==I;
      );
      O(;
      L     #Wpis._3_dbb13_Kod_Maszyna;
      L     #Wpis.Kod_Spr_KB2;
      ==I;
      );
      O(;
      L     #Wpis._3_dbb13_Kod_Maszyna;
      L     #Wpis.Kod_Spr_I1;
      ==I;
      );
      O(;
      L     #Wpis._3_dbb13_Kod_Maszyna;
      L     #Wpis.Kod_Spr_I2;
      ==I;
      );
      O(;
      L     #Wpis._3_dbb13_Kod_Maszyna;
      L     #Wpis.Kod_Spr_I3;
      ==I;
      );
      JC    d_12;
      L     0;
      T     #Wpis._3_dbb12_Kod_Kier;
      T     #Wpis._3_dbb13_Kod_Maszyna;
      T     #Wpis._3_dbw14_War_Wagowa;
d_12: NOP   0;
//Przeprowadzeni sprwdzenia   dbd 16 (pozycja 5)
      O(;
      L     #Wpis._4_dbb17_Kod_Maszyna;
      L     #Wpis.Kod_Spr_KB1;
      ==I;
      );
      O(;
      L     #Wpis._4_dbb17_Kod_Maszyna;
      L     #Wpis.Kod_Spr_KB2;
      ==I;
      );
      O(;
      L     #Wpis._4_dbb17_Kod_Maszyna;
      L     #Wpis.Kod_Spr_I1;
      ==I;
      );
      O(;
      L     #Wpis._4_dbb17_Kod_Maszyna;
      L     #Wpis.Kod_Spr_I2;
      ==I;
      );
      O(;
      L     #Wpis._4_dbb17_Kod_Maszyna;
      L     #Wpis.Kod_Spr_I3;
      ==I;
      );
      JC    d_16;
      L     0;
      T     #Wpis._4_dbb16_Kod_Kier;
      T     #Wpis._4_dbb17_Kod_Maszyna;
      T     #Wpis._4_dbw18_War_Wagowa;
d_16: NOP   0;
NETWORK
TITLE =
//Kasowanie zer w rejestrze. Polega na przesuwaniu wszystkiego w gore i tym samym 
//luki sa wycinane.Gdy zniknie paleta stos wycina element i przsuwa reszte w 
//gore.
//**********Pozycja 12.0
      L     LD 12;
      L     0;
      ==D;
      JCN   o1;
      L     LD 16;
      T     LD 12;
      L     LD 20;
      T     LD 16;
      L     LD 24;
      T     LD 20;
      L     LD 28;
      T     LD 24;
      L     LD 32;
      T     LD 28;
o1:   NOP   0;
//**********Pozycja 16.0
      L     LD 16;
      L     0;
      ==D;
      JCN   o2;
      L     LD 20;
      T     LD 16;
      L     LD 24;
      T     LD 20;
      L     LD 28;
      T     LD 24;
      L     LD 32;
      T     LD 28;
o2:   NOP   0;
//**********Pozycja 20.0
      L     LD 20;
      L     0;
      ==D;
      JCN   o3;
      L     LD 24;
      T     LD 20;
      L     LD 28;
      T     LD 24;
      L     LD 32;
      T     LD 28;
o3:   NOP   0;
//**********Pozycja 24.0
      L     LD 24;
      L     0;
      ==D;
      JCN   o4;
      L     LD 28;
      T     LD 24;
      L     LD 32;
      T     LD 28;
o4:   NOP   0;
//**********Pozycja 28.0
      L     LD 28;
      L     0;
      ==D;
      JCN   o5;
      L     LD 32;
      T     LD 28;
o5:   NOP   0;
NETWORK
TITLE =
//Zaladowanie nowej wartosci do KB1
//Wyresetuj bity tymczasowe
      SET;
      R     #Temp_Wpis_KB1;
      R     #Temp_Wpis_KB2;
      R     #Temp_Wpis_I1;
      R     #Temp_Wpis_I2;
      R     #Temp_Wpis_I3;
      A     #P.KB1_Istnieje;
      AN    #P.KB1_Wpis;
      JCN   z0;
      L     #id_Wartosc_KB1;
      T     #Help_Dint;
      AN    #P.KB1_Wpis;
      =     #Temp_Wpis_KB1;
      JU    x0;
z0:   NOP   0;
      A     #P.KB2_Istnieje;
      AN    #P.KB2_Wpis;
      JCN   z1;
      L     #id_Wartosc_KB2;
      T     #Help_Dint;
      AN    #P.KB2_Wpis;
      =     #Temp_Wpis_KB2;
      JU    x0;
z1:   NOP   0;
      A     #P.I1_Istnieje;
      AN    #P.I1_Wpis;
      JCN   z2;
      L     #id_Wartosc_I1;
      T     #Help_Dint;
      AN    #P.I1_Wpis;
      =     #Temp_Wpis_I1;
      JU    x0;
z2:   NOP   0;
      A     #P.I2_Istnieje;
      AN    #P.I2_Wpis;
      JCN   z3;
      L     #id_Wartosc_I2;
      T     #Help_Dint;
      AN    #P.I2_Wpis;
      =     #Temp_Wpis_I2;
      JU    x0;
z3:   NOP   0;
      A     #P.I3_Istnieje;
      AN    #P.I3_Wpis;
      JCN   z4;
      L     #id_Wartosc_I3;
      T     #Help_Dint;
      AN    #P.I3_Wpis;
      =     #Temp_Wpis_I3;
      JU    x0;
z4:   NOP   0;
//wartosc wagowa
//***sprawdzenie pozycji 0**********************
x0:   L     LW 10;
      L     #Wpis._0_dbw2_War_Wagowa;
      >I;
      A(;
      O     #Temp_Wpis_KB1;
      O     #Temp_Wpis_KB2;
      O     #Temp_Wpis_I1;
      O     #Temp_Wpis_I2;
      O     #Temp_Wpis_I3;
      );
      JCN   k0;
//zrobienie miejsca na nowy rekord
//***pozycja 4-5
      L     LD 28;
      T     LD 32;
//***pozycja 3-4
      L     LD 24;
      T     LD 28;
//***pozycja 2-3
      L     LD 20;
      T     LD 24;
//***pozycja 1-2
      L     LD 16;
      T     LD 20;
//***pozycja 0-1
      L     LD 12;
      T     LD 16;
      L     #Help_Dint;	//id_wartosc
      T     LD 12;	//element
//Potwierdzenie wpisania
      A     #Temp_Wpis_KB1;
      S     #P.KB1_Wpis;
      A     #Temp_Wpis_KB2;
      S     #P.KB2_Wpis;
      A     #Temp_Wpis_I1;
      S     #P.I1_Wpis;
      A     #Temp_Wpis_I2;
      S     #P.I2_Wpis;
      A     #Temp_Wpis_I3;
      S     #P.I3_Wpis;
      SET;
      R     #Temp_Wpis_KB1;
      R     #Temp_Wpis_KB2;
      R     #Temp_Wpis_I1;
      R     #Temp_Wpis_I2;
      R     #Temp_Wpis_I3;
k0:   NOP   0;
//***sprawdzenie pozycji 1**********************
      L     LW 10;
      L     #Wpis._1_dbw6_War_Wagowa;
      >I;
      A(;
      O     #Temp_Wpis_KB1;
      O     #Temp_Wpis_KB2;
      O     #Temp_Wpis_I1;
      O     #Temp_Wpis_I2;
      O     #Temp_Wpis_I3;
      );
      JCN   k1;
//***pozycja 4-5
      L     LD 28;
      T     LD 32;
//***pozycja 3-4
      L     LD 24;
      T     LD 28;
//***pozycja 2-3
      L     LD 20;
      T     LD 24;
//***pozycja 1-2
      L     LD 16;
      T     LD 20;
      L     #Help_Dint;	//id_wartosc
      T     LD 16;	//element
//Potwierdzenie wpisania
      A     #Temp_Wpis_KB1;
      S     #P.KB1_Wpis;
      A     #Temp_Wpis_KB2;
      S     #P.KB2_Wpis;
      A     #Temp_Wpis_I1;
      S     #P.I1_Wpis;
      A     #Temp_Wpis_I2;
      S     #P.I2_Wpis;
      A     #Temp_Wpis_I3;
      S     #P.I3_Wpis;
      SET;
      R     #Temp_Wpis_KB1;
      R     #Temp_Wpis_KB2;
      R     #Temp_Wpis_I1;
      R     #Temp_Wpis_I2;
      R     #Temp_Wpis_I3;
k1:   NOP   0;
//***sprawdzenie pozycji 2
      L     LW 10;
      L     #Wpis._2_dbw10_War_Wagowa;
      >I;
      A(;
      O     #Temp_Wpis_KB1;
      O     #Temp_Wpis_KB2;
      O     #Temp_Wpis_I1;
      O     #Temp_Wpis_I2;
      O     #Temp_Wpis_I3;
      );
      JCN   k2;
//***pozycja 4-5
      L     LD 28;
      T     LD 32;
//***pozycja 3-4
      L     LD 24;
      T     LD 28;
//***pozycja 2-3
      L     LD 20;
      T     LD 24;
      L     #Help_Dint;	//id_wartosc
      T     LD 20;	//element
//Potwierdzenie wpisania
      A     #Temp_Wpis_KB1;
      S     #P.KB1_Wpis;
      A     #Temp_Wpis_KB2;
      S     #P.KB2_Wpis;
      A     #Temp_Wpis_I1;
      S     #P.I1_Wpis;
      A     #Temp_Wpis_I2;
      S     #P.I2_Wpis;
      A     #Temp_Wpis_I3;
      S     #P.I3_Wpis;
      SET;
      R     #Temp_Wpis_KB1;
      R     #Temp_Wpis_KB2;
      R     #Temp_Wpis_I1;
      R     #Temp_Wpis_I2;
      R     #Temp_Wpis_I3;
k2:   NOP   0;
//***sprawdzenie pozycji 3
      L     LW 10;
      L     #Wpis._3_dbw14_War_Wagowa;
      >I;
      A(;
      O     #Temp_Wpis_KB1;
      O     #Temp_Wpis_KB2;
      O     #Temp_Wpis_I1;
      O     #Temp_Wpis_I2;
      O     #Temp_Wpis_I3;
      );
      JCN   k3;
//***pozycja 4-5
      L     LD 28;
      T     LD 32;
//***pozycja 3-4
      L     LD 24;
      T     LD 28;
      L     #Help_Dint;	//id_wartosc
      T     LD 24;	//element
//Potwierdzenie wpisania
      A     #Temp_Wpis_KB1;
      S     #P.KB1_Wpis;
      A     #Temp_Wpis_KB2;
      S     #P.KB2_Wpis;
      A     #Temp_Wpis_I1;
      S     #P.I1_Wpis;
      A     #Temp_Wpis_I2;
      S     #P.I2_Wpis;
      A     #Temp_Wpis_I3;
      S     #P.I3_Wpis;
      SET;
      R     #Temp_Wpis_KB1;
      R     #Temp_Wpis_KB2;
      R     #Temp_Wpis_I1;
      R     #Temp_Wpis_I2;
      R     #Temp_Wpis_I3;
k3:   NOP   0;
//***sprawdzenie pozycji 4
      L     LW 10;
      L     #Wpis._4_dbw18_War_Wagowa;
      >I;
      A(;
      O     #Temp_Wpis_KB1;
      O     #Temp_Wpis_KB2;
      O     #Temp_Wpis_I1;
      O     #Temp_Wpis_I2;
      O     #Temp_Wpis_I3;
      );
      JCN   k4;
//***pozycja 4-5
      L     LD 28;
      T     LD 32;
      L     #Help_Dint;	//id_wartosc
      T     LD 28;	//element
//Potwierdzenie wpisania
      A     #Temp_Wpis_KB1;
      S     #P.KB1_Wpis;
      A     #Temp_Wpis_KB2;
      S     #P.KB2_Wpis;
      A     #Temp_Wpis_I1;
      S     #P.I1_Wpis;
      A     #Temp_Wpis_I2;
      S     #P.I2_Wpis;
      A     #Temp_Wpis_I3;
      S     #P.I3_Wpis;
      SET;
      R     #Temp_Wpis_KB1;
      R     #Temp_Wpis_KB2;
      R     #Temp_Wpis_I1;
      R     #Temp_Wpis_I2;
      R     #Temp_Wpis_I3;
k4:   NOP   0;
//***sprawdzenie pozycji 5
      L     LW 10;
      L     #Wpis._5_dbw22_War_Wagowa;
      >I;
      A(;
      O     #Temp_Wpis_KB1;
      O     #Temp_Wpis_KB2;
      O     #Temp_Wpis_I1;
      O     #Temp_Wpis_I2;
      O     #Temp_Wpis_I3;
      );
      JCN   k5;
//***pozycja 4-5
      L     #Help_Dint;	//id_wartosc
      T     LD 32;	//element
//Potwierdzenie wpisania
      A     #Temp_Wpis_KB1;
      S     #P.KB1_Wpis;
      A     #Temp_Wpis_KB2;
      S     #P.KB2_Wpis;
      A     #Temp_Wpis_I1;
      S     #P.I1_Wpis;
      A     #Temp_Wpis_I2;
      S     #P.I2_Wpis;
      A     #Temp_Wpis_I3;
      S     #P.I3_Wpis;
      SET;
      R     #Temp_Wpis_KB1;
      R     #Temp_Wpis_KB2;
      R     #Temp_Wpis_I1;
      R     #Temp_Wpis_I2;
      R     #Temp_Wpis_I3;
k5:   NOP   0;
NETWORK
TITLE =
NETWORK
TITLE =
//Sprawdzenie czy wpisy nie sa zerami
      L     #Wpis._0_dbw2_War_Wagowa;
      L     0;
      >I;
      =     #P.Wpis_0_istnieje;
//1
      L     #Wpis._1_dbw6_War_Wagowa;
      L     0;
      >I;
      =     #P.Wpis_1_istnieje;
//2
      L     #Wpis._2_dbw10_War_Wagowa;
      L     0;
      >I;
      =     #P.Wpis_2_istnieje;
//3
      L     #Wpis._3_dbw14_War_Wagowa;
      L     0;
      >I;
      =     #P.Wpis_3_istnieje;
//4
      L     #Wpis._4_dbw18_War_Wagowa;
      L     0;
      >I;
      =     #P.Wpis_4_istnieje;
//5
      L     #Wpis._5_dbw22_War_Wagowa;
      L     0;
      >I;
      =     #P.Wpis_5_istnieje;
NETWORK
TITLE =
//Przesowanie rejestrow w gore i dol
//toggle 0 i 1 
      A(;
      O     #i_Poz_5_Down;
      O     #i_Poz_4_Up;
      );
      FP    #P.edge_1;
      A     #P.Wpis_0_istnieje;
      A     #P.Wpis_1_istnieje;
      JCN   w0;
      L     LW 12;
      T     #Help_Int_2;
      L     #Wpis._0_dbw2_War_Wagowa;
      T     LW 12;
      L     #Help_Int_2;
      T     #Wpis._0_dbw2_War_Wagowa;
w0:   NOP   0;
//toggle 1 i 2  
      A(;
      O     #i_Poz_4_Down;
      O     #i_Poz_3_Up;
      );
      FP    #P.edge_2;
      A     #P.Wpis_1_istnieje;
      A     #P.Wpis_2_istnieje;
      JCN   w1;
      L     #Wpis._0_dbw2_War_Wagowa;
      T     #Help_Int_2;
      L     #Wpis._1_dbw6_War_Wagowa;
      T     #Wpis._0_dbw2_War_Wagowa;
      L     #Help_Int_2;
      T     #Wpis._1_dbw6_War_Wagowa;
w1:   NOP   0;
//toggle 2 i 3  
      A(;
      O     #i_Poz_3_Down;
      O     #i_Poz_2_Up;
      );
      FP    #P.edge_3;
      A     #P.Wpis_2_istnieje;
      A     #P.Wpis_3_istnieje;
      JCN   w2;
      L     #Wpis._1_dbw6_War_Wagowa;
      T     #Help_Int_2;
      L     #Wpis._2_dbw10_War_Wagowa;
      T     #Wpis._1_dbw6_War_Wagowa;
      L     #Help_Int_2;
      T     #Wpis._2_dbw10_War_Wagowa;
w2:   NOP   0;
//toggle 3 i 4  
      A(;
      O     #i_Poz_2_Down;
      O     #i_Poz_1_Up;
      );
      FP    #P.edge_4;
      A     #P.Wpis_3_istnieje;
      A     #P.Wpis_4_istnieje;
      JCN   w3;
      L     #Wpis._2_dbw10_War_Wagowa;
      T     #Help_Int_2;
      L     #Wpis._3_dbw14_War_Wagowa;
      T     #Wpis._2_dbw10_War_Wagowa;
      L     #Help_Int_2;
      T     #Wpis._3_dbw14_War_Wagowa;
w3:   NOP   0;
NETWORK
TITLE =
      L     #P;
      T     #iow_Help_DWord;
//Zaladowanie pakietu danych
      CALL  "BLKMOV" (
           SRCBLK                   := #Wpis,
           RET_VAL                  := #Help_Blok_Move,
           DSTBLK                   := "Key_DB".Wpis);
END_FUNCTION

FUNCTION "Wozek_Jezdny_Kolejka" : VOID	// FC 600
//Nalezy w HMI dopisac brakujace kody obslugi jazdy (kod 17 i kod 18)
//
VERSION : 0.1
BEGIN
NETWORK
TITLE =
//Ten Network celowo jest wolny
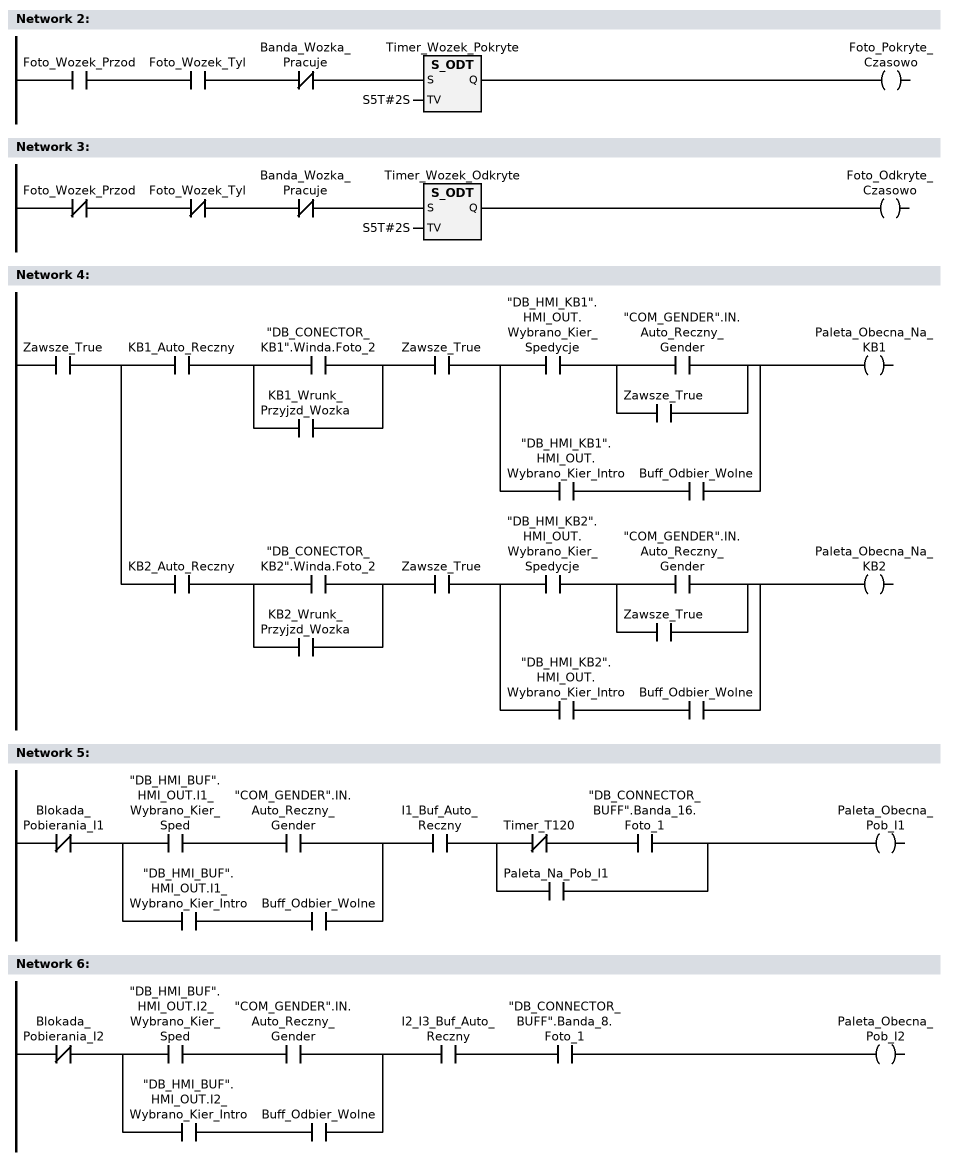
NETWORK
TITLE =
//Fotokomorki pokryte  i silnik band nie pracuje
      A     "Foto_Wozek_Przod";
      A     "Foto_Wozek_Tyl";
      AN    "Banda_Wozka_Pracuje";
      L     S5T#2S;
      SD    "Timer_Wozek_Pokryte";
      NOP   0;
      NOP   0;
      NOP   0;
      A     "Timer_Wozek_Pokryte";
      =     "Foto_Pokryte_Czasowo";
NETWORK
TITLE =
      AN    "Foto_Wozek_Przod";
      AN    "Foto_Wozek_Tyl";
      AN    "Banda_Wozka_Pracuje";
      L     S5T#2S;
      SD    "Timer_Wozek_Odkryte";
      NOP   0;
      NOP   0;
      NOP   0;
      A     "Timer_Wozek_Odkryte";
      =     "Foto_Odkryte_Czasowo";
NETWORK
TITLE =
//Sprawdznie Czy paleta jest gotowa do odebrania
//-Dodanie warunku Gender w automacie na przejazd na Gender db205.dbx0.1
      A     "Zawsze_True";
      =     L 0.0;
      A     L 0.0;
      A     "KB1_Auto_Reczny";
      A(;
      O     "DB_CONECTOR_KB1".Winda.Foto_2;
      O     "KB1_Wrunk_Przyjzd_Wozka";
      );
      A     "Zawsze_True";
      A(;
      A     "DB_HMI_KB1".HMI_OUT.Wybrano_Kier_Spedycje;
      A(;
      O     "COM_GENDER".IN.Auto_Reczny_Gender;
      O     "Zawsze_True";
      );
      O;
      A     "DB_HMI_KB1".HMI_OUT.Wybrano_Kier_Intro;
      A     "Buff_Odbier_Wolne";
      );
      =     "Paleta_Obecna_Na_KB1";
      A     L 0.0;
      A     "KB2_Auto_Reczny";
      A(;
      O     "DB_CONECTOR_KB2".Winda.Foto_2;
      O     "KB2_Wrunk_Przyjzd_Wozka";
      );
      A     "Zawsze_True";
      A(;
      A     "DB_HMI_KB2".HMI_OUT.Wybrano_Kier_Spedycje;
      A(;
      O     "COM_GENDER".IN.Auto_Reczny_Gender;
      O     "Zawsze_True";
      );
      O;
      A     "DB_HMI_KB2".HMI_OUT.Wybrano_Kier_Intro;
      A     "Buff_Odbier_Wolne";
      );
      =     "Paleta_Obecna_Na_KB2";
NETWORK
TITLE =
      AN    "Blokada_Pobierania_I1";
      A(;
      A     "DB_HMI_BUF".HMI_OUT.I1_Wybrano_Kier_Sped;
      A     "COM_GENDER".IN.Auto_Reczny_Gender;
      O;
      A     "DB_HMI_BUF".HMI_OUT.I1_Wybrano_Kier_Intro;
      A     "Buff_Odbier_Wolne";
      );
      A     "I1_Buf_Auto_Reczny";
      A(;
      AN    "Timer_T120";
      A     "DB_CONNECTOR_BUFF".Banda_16.Foto_1;
      O     "Paleta_Na_Pob_I1";
      );
      =     "Paleta_Obecna_Pob_I1";
NETWORK
TITLE =
//Blokowanie pobierania palet na I2
      AN    "Blokada_Pobierania_I2";
      A(;
      A     "DB_HMI_BUF".HMI_OUT.I2_Wybrano_Kier_Sped;
      A     "COM_GENDER".IN.Auto_Reczny_Gender;
      O;
      A     "DB_HMI_BUF".HMI_OUT.I2_Wybrano_Kier_Intro;
      A     "Buff_Odbier_Wolne";
      );
      A     "I2_I3_Buf_Auto_Reczny";
      A     "DB_CONNECTOR_BUFF".Banda_8.Foto_1;
      =     "Paleta_Obecna_Pob_I2";
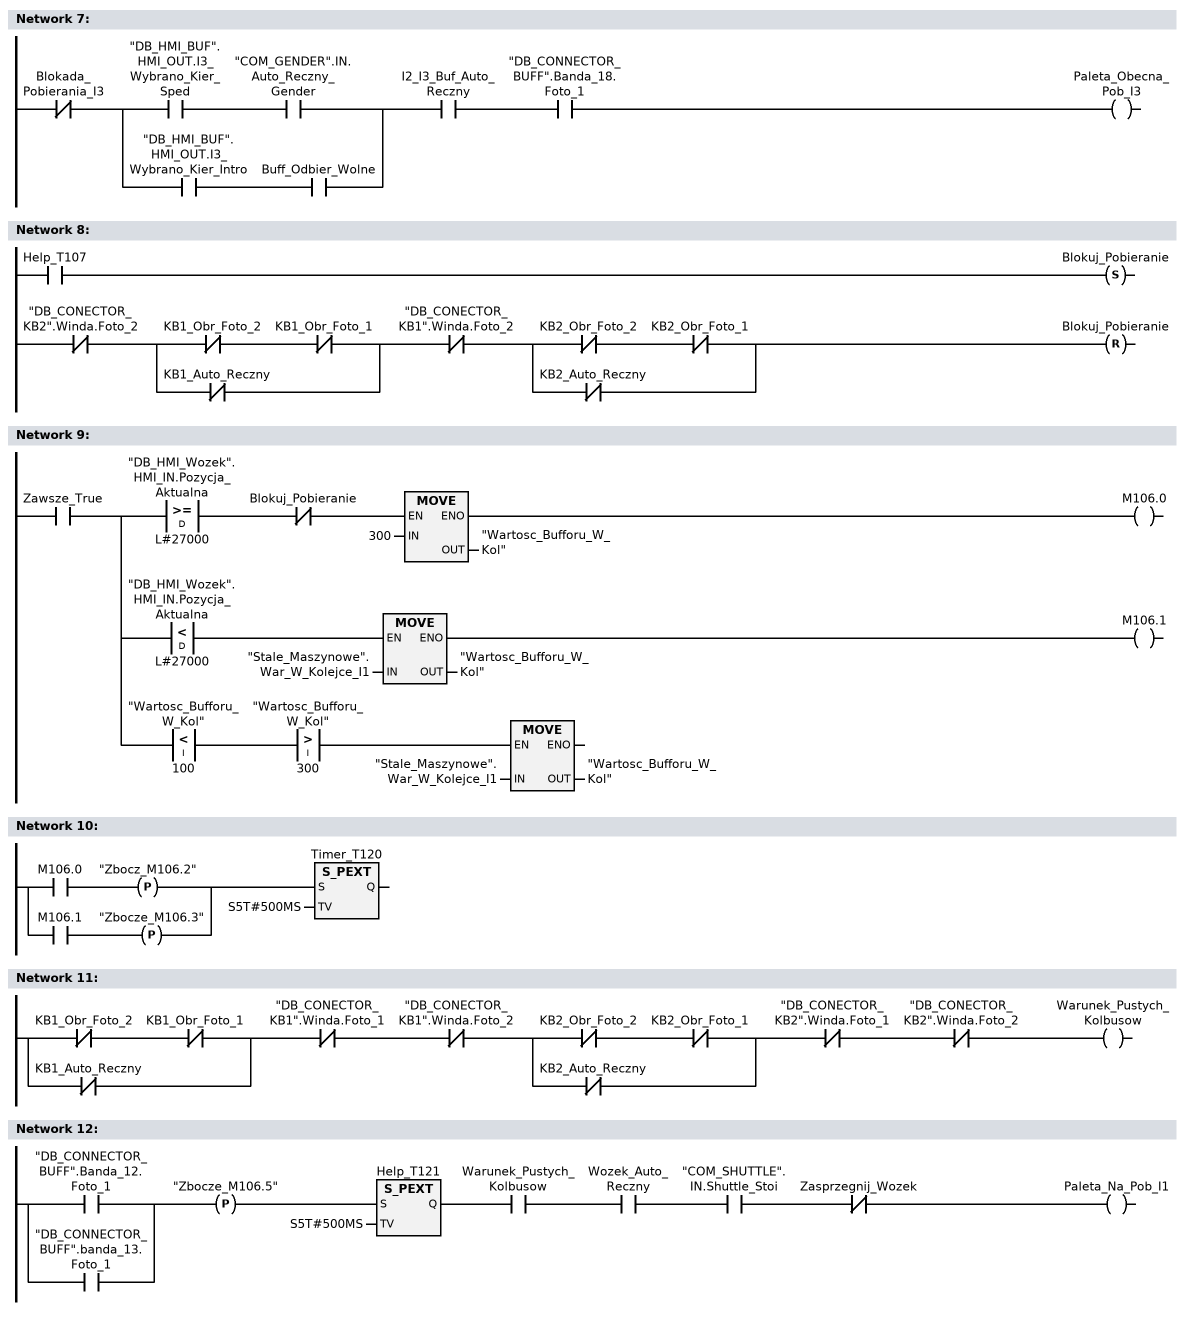
NETWORK
TITLE =
//Blokowanie pobierania palet na I3
      AN    "Blokada_Pobierania_I3";
      A(;
      A     "DB_HMI_BUF".HMI_OUT.I3_Wybrano_Kier_Sped;
      A     "COM_GENDER".IN.Auto_Reczny_Gender;
      O;
      A     "DB_HMI_BUF".HMI_OUT.I3_Wybrano_Kier_Intro;
      A     "Buff_Odbier_Wolne";
      );
      A     "I2_I3_Buf_Auto_Reczny";
      A     "DB_CONNECTOR_BUFF".Banda_18.Foto_1;
      =     "Paleta_Obecna_Pob_I3";
NETWORK
TITLE =
//Gdy wcisniety przycisk Reset to najpierw pobiera palety z kolbusow
      A     "Help_T107";
      S     "Blokuj_Pobieranie";
      AN    "DB_CONECTOR_KB2".Winda.Foto_2;
      A(;
      AN    "KB1_Obr_Foto_2";
      AN    "KB1_Obr_Foto_1";
      ON    "KB1_Auto_Reczny";
      );
      AN    "DB_CONECTOR_KB1".Winda.Foto_2;
      A(;
      AN    "KB2_Obr_Foto_2";
      AN    "KB2_Obr_Foto_1";
      ON    "KB2_Auto_Reczny";
      );
      R     "Blokuj_Pobieranie";
      NOP   0;
NETWORK
TITLE =
//Zeby wozek cofnal sie do pobierania gdy oddaje palete na buffor
      A     "Zawsze_True";
      =     L 0.0;
      A     L 0.0;
      A(;
      L     "DB_HMI_Wozek".HMI_IN.Pozycja_Aktualna;
      L     L#27000;
      >=D;
      );
      AN    "Blokuj_Pobieranie";
      JNB   _001;
      L     300;
      T     "Wartosc_Bufforu_W_Kol";
      SET;
      SAVE;
      CLR;
_001: A     BR;
      =     "M106.0";
      A     L 0.0;
      A(;
      L     "DB_HMI_Wozek".HMI_IN.Pozycja_Aktualna;
      L     L#27000;
      <D;
      );
      JNB   _002;
      L     "Stale_Maszynowe".War_W_Kolejce_I1;
      T     "Wartosc_Bufforu_W_Kol";
      SET;
      SAVE;
      CLR;
_002: A     BR;
      =     "M106.1";
      A     L 0.0;
      A(;
      L     "Wartosc_Bufforu_W_Kol";
      L     100;
      <I;
      );
      A(;
      L     "Wartosc_Bufforu_W_Kol";
      L     300;
      >I;
      );
      JNB   _003;
      L     "Stale_Maszynowe".War_W_Kolejce_I1;
      T     "Wartosc_Bufforu_W_Kol";
_003: NOP   0;
NETWORK
TITLE =
//Aby bylo cofanie sie na buffor jak juz jest blisko
      A(;
      A     "M106.0";
      FP    "Zbocz_M106.2";
      O(;
      A     "M106.1";
      FP    "Zbocze_M106.3";
      );
      );
      L     S5T#500MS;
      SE    "Timer_T120";
      NOP   0;
      NOP   0;
      NOP   0;
      NOP   0;
NETWORK
TITLE =
//Algorytm jazdy spec. intro
      A(;
      AN    "KB1_Obr_Foto_2";
      AN    "KB1_Obr_Foto_1";
      ON    "KB1_Auto_Reczny";
      );
      AN    "DB_CONECTOR_KB1".Winda.Foto_1;
      AN    "DB_CONECTOR_KB1".Winda.Foto_2;
      A(;
      AN    "KB2_Obr_Foto_2";
      AN    "KB2_Obr_Foto_1";
      ON    "KB2_Auto_Reczny";
      );
      AN    "DB_CONECTOR_KB2".Winda.Foto_1;
      AN    "DB_CONECTOR_KB2".Winda.Foto_2;
      =     "Warunek_Pustych_Kolbusow";
NETWORK
TITLE =
      A(;
      A(;
      O     "DB_CONNECTOR_BUFF".Banda_12.Foto_1;
      O     "DB_CONNECTOR_BUFF".banda_13.Foto_1;
      );
      FP    "Zbocze_M106.5";
      L     S5T#500MS;
      SE    "Help_T121";
      NOP   0;
      NOP   0;
      NOP   0;
      A     "Help_T121";
      );
      A     "Warunek_Pustych_Kolbusow";
      A     "Wozek_Auto_Reczny";
      A     "COM_SHUTTLE".IN.Shuttle_Stoi;
      AN    "Zasprzegnij_Wozek";
      =     "Paleta_Na_Pob_I1";
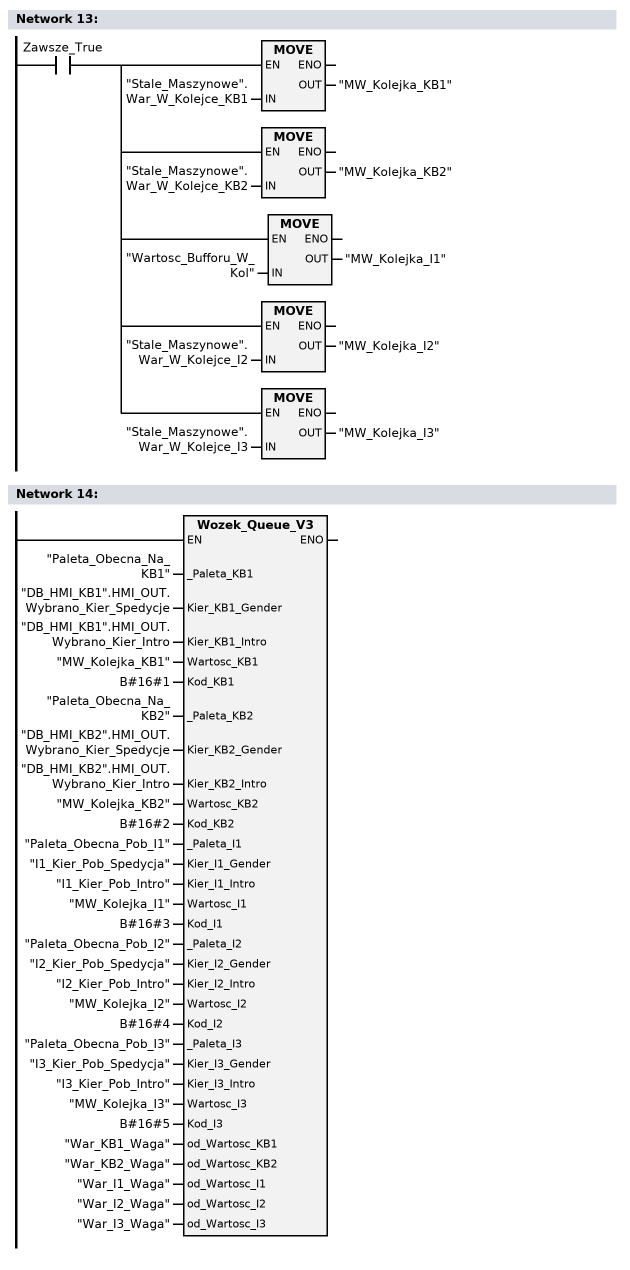
NETWORK
TITLE =
//Wartosc danej pozycji w kolejce
      A     "Zawsze_True";
      =     L 0.0;
      A     L 0.0;
      JNB   _004;
      L     "Stale_Maszynowe".War_W_Kolejce_KB1;
      T     "MW_Kolejka_KB1";
_004: NOP   0;
      A     L 0.0;
      JNB   _005;
      L     "Stale_Maszynowe".War_W_Kolejce_KB2;
      T     "MW_Kolejka_KB2";
_005: NOP   0;
      A     L 0.0;
      JNB   _006;
      L     "Wartosc_Bufforu_W_Kol";
      T     "MW_Kolejka_I1";
_006: NOP   0;
      A     L 0.0;
      JNB   _007;
      L     "Stale_Maszynowe".War_W_Kolejce_I2;
      T     "MW_Kolejka_I2";
_007: NOP   0;
      A     L 0.0;
      JNB   _008;
      L     "Stale_Maszynowe".War_W_Kolejce_I3;
      T     "MW_Kolejka_I3";
_008: NOP   0;
NETWORK
TITLE =
//Dostep do kolejki jazdy wozkiem
//MB620-kierunek intro(0),spedycja(1)
//MB621-Kod mszyny np KB1-1
//MW622-Wartosc wagowa (Pobrana ze stalych maszynowych)
//
//
//
      CALL  "Wozek_Queue_V3" (
           _Paleta_KB1              := "Paleta_Obecna_Na_KB1",
           Kier_KB1_Gender          := "DB_HMI_KB1".HMI_OUT.Wybrano_Kier_Spedycje,
           Kier_KB1_Intro           := "DB_HMI_KB1".HMI_OUT.Wybrano_Kier_Intro,
           Wartosc_KB1              := "MW_Kolejka_KB1",
           Kod_KB1                  := B#16#1,
           _Paleta_KB2              := "Paleta_Obecna_Na_KB2",
           Kier_KB2_Gender          := "DB_HMI_KB2".HMI_OUT.Wybrano_Kier_Spedycje,
           Kier_KB2_Intro           := "DB_HMI_KB2".HMI_OUT.Wybrano_Kier_Intro,
           Wartosc_KB2              := "MW_Kolejka_KB2",
           Kod_KB2                  := B#16#2,
           _Paleta_I1               := "Paleta_Obecna_Pob_I1",
           Kier_I1_Gender           := "I1_Kier_Pob_Spedycja",
           Kier_I1_Intro            := "I1_Kier_Pob_Intro",
           Wartosc_I1               := "MW_Kolejka_I1",
           Kod_I1                   := B#16#3,
           _Paleta_I2               := "Paleta_Obecna_Pob_I2",
           Kier_I2_Gender           := "I2_Kier_Pob_Spedycja",
           Kier_I2_Intro            := "I2_Kier_Pob_Intro",
           Wartosc_I2               := "MW_Kolejka_I2",
           Kod_I2                   := B#16#4,
           _Paleta_I3               := "Paleta_Obecna_Pob_I3",
           Kier_I3_Gender           := "I3_Kier_Pob_Spedycja",
           Kier_I3_Intro            := "I3_Kier_Pob_Intro",
           Wartosc_I3               := "MW_Kolejka_I3",
           Kod_I3                   := B#16#5,
           od_Wartosc_KB1           := "War_KB1_Waga",
           od_Wartosc_KB2           := "War_KB2_Waga",
           od_Wartosc_I1            := "War_I1_Waga",
           od_Wartosc_I2            := "War_I2_Waga",
           od_Wartosc_I3            := "War_I3_Waga");
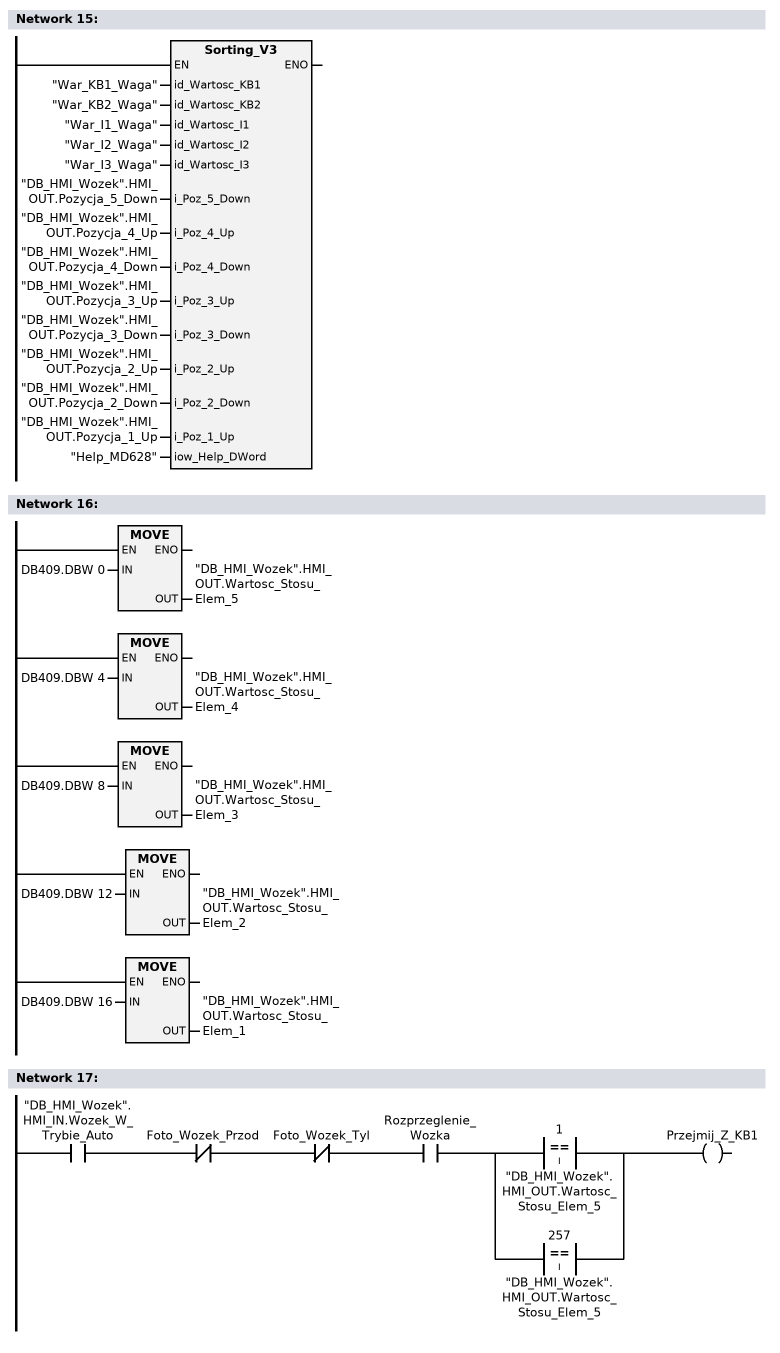
NETWORK
TITLE =
//Zbudowanie rekordu
      CALL  "Sorting_V3" (
           id_Wartosc_KB1           := "War_KB1_Waga",
           id_Wartosc_KB2           := "War_KB2_Waga",
           id_Wartosc_I1            := "War_I1_Waga",
           id_Wartosc_I2            := "War_I2_Waga",
           id_Wartosc_I3            := "War_I3_Waga",
           i_Poz_5_Down             := "DB_HMI_Wozek".HMI_OUT.Pozycja_5_Down,
           i_Poz_4_Up               := "DB_HMI_Wozek".HMI_OUT.Pozycja_4_Up,
           i_Poz_4_Down             := "DB_HMI_Wozek".HMI_OUT.Pozycja_4_Down,
           i_Poz_3_Up               := "DB_HMI_Wozek".HMI_OUT.Pozycja_3_Up,
           i_Poz_3_Down             := "DB_HMI_Wozek".HMI_OUT.Pozycja_3_Down,
           i_Poz_2_Up               := "DB_HMI_Wozek".HMI_OUT.Pozycja_2_Up,
           i_Poz_2_Down             := "DB_HMI_Wozek".HMI_OUT.Pozycja_2_Down,
           i_Poz_1_Up               := "DB_HMI_Wozek".HMI_OUT.Pozycja_1_Up,
           iow_Help_DWord           := "Help_MD628");
NETWORK
TITLE =
//Wyswietlenie pozycji na HMI
//Mozliwe kombinacje:
//001-KB1-intro
//101-KB1-spedycja
//002-KB2-intro
//102-KB2-spedycja
//003-i1-intro odbieranie
//103-i1-spedycja
//004-i2-intro odbieranie
//104-i2-spedycja
//005-i3-intro odbieranie
//105-i3-spedycja
//Przypisanie wartosci do wizualizacji
      L     DB409.DBW 0;
      T     "DB_HMI_Wozek".HMI_OUT.Wartosc_Stosu_Elem_5;
      L     DB409.DBW 4;
      T     "DB_HMI_Wozek".HMI_OUT.Wartosc_Stosu_Elem_4;
      L     DB409.DBW 8;
      T     "DB_HMI_Wozek".HMI_OUT.Wartosc_Stosu_Elem_3;
      L     DB409.DBW 12;
      T     "DB_HMI_Wozek".HMI_OUT.Wartosc_Stosu_Elem_2;
      L     DB409.DBW 16;
      T     "DB_HMI_Wozek".HMI_OUT.Wartosc_Stosu_Elem_1;
NETWORK
TITLE =
//Wozek jest w automatyce. Przejmij palete z KB1
      A     "DB_HMI_Wozek".HMI_IN.Wozek_W_Trybie_Auto;
      AN    "Foto_Wozek_Przod";
      AN    "Foto_Wozek_Tyl";
      A     "Rozprzeglenie_Wozka";
      A(;
      O(;
      L     1;
      L     "DB_HMI_Wozek".HMI_OUT.Wartosc_Stosu_Elem_5;
      ==I;
      );
      O(;
      L     257;
      L     "DB_HMI_Wozek".HMI_OUT.Wartosc_Stosu_Elem_5;
      ==I;
      );
      );
      =     "Przejmij_Z_KB1";
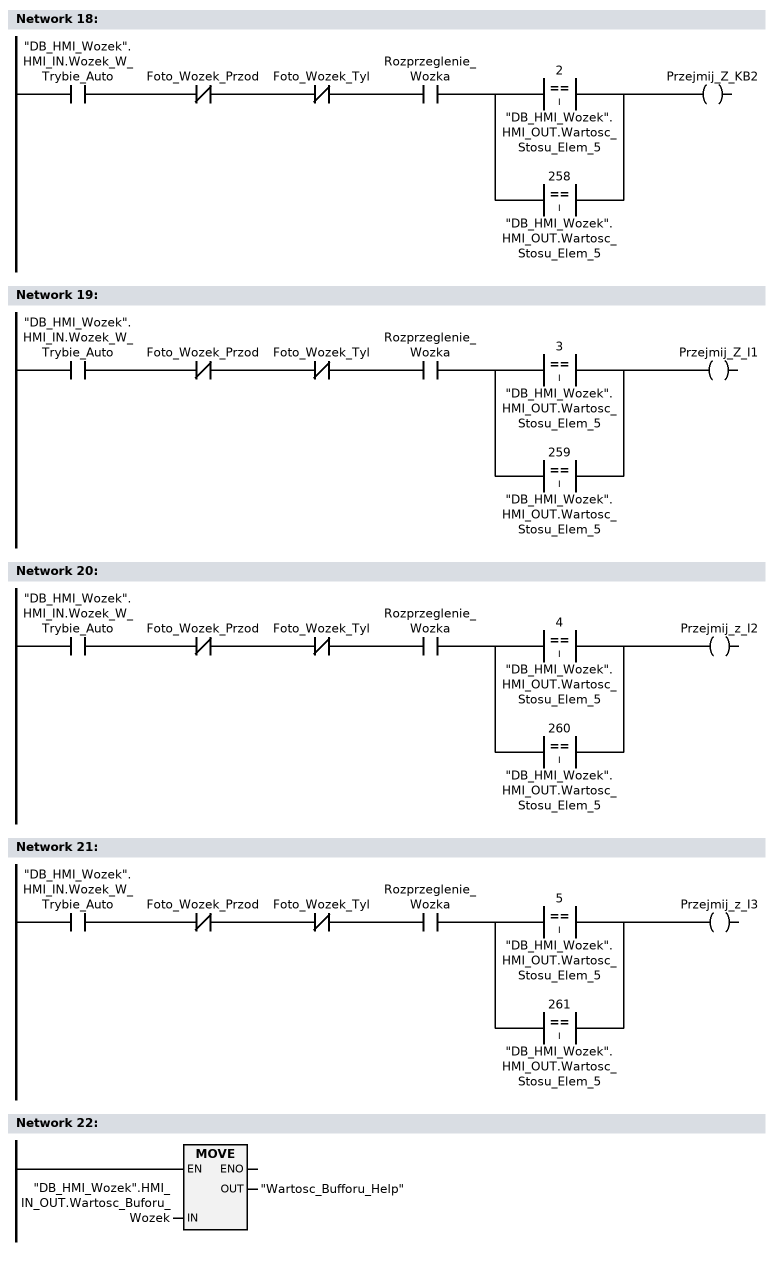
NETWORK
TITLE =
//Wozek jest w automatyce. Przejmij palete z KB2
//
      A     "DB_HMI_Wozek".HMI_IN.Wozek_W_Trybie_Auto;
      AN    "Foto_Wozek_Przod";
      AN    "Foto_Wozek_Tyl";
      A     "Rozprzeglenie_Wozka";
      A(;
      O(;
      L     2;
      L     "DB_HMI_Wozek".HMI_OUT.Wartosc_Stosu_Elem_5;
      ==I;
      );
      O(;
      L     258;
      L     "DB_HMI_Wozek".HMI_OUT.Wartosc_Stosu_Elem_5;
      ==I;
      );
      );
      =     "Przejmij_Z_KB2";
NETWORK
TITLE =
//Wozek jest w automatyce. Przejmij palete z intro 1
//
      A     "DB_HMI_Wozek".HMI_IN.Wozek_W_Trybie_Auto;
      AN    "Foto_Wozek_Przod";
      AN    "Foto_Wozek_Tyl";
      A     "Rozprzeglenie_Wozka";
      A(;
      O(;
      L     3;
      L     "DB_HMI_Wozek".HMI_OUT.Wartosc_Stosu_Elem_5;
      ==I;
      );
      O(;
      L     259;
      L     "DB_HMI_Wozek".HMI_OUT.Wartosc_Stosu_Elem_5;
      ==I;
      );
      );
      =     "Przejmij_Z_I1";
NETWORK
TITLE =
//Przejmij paleta z intro 2  (260!!!!!!!!!!!!!!!!!!!!!!)
      A     "DB_HMI_Wozek".HMI_IN.Wozek_W_Trybie_Auto;
      AN    "Foto_Wozek_Przod";
      AN    "Foto_Wozek_Tyl";
      A     "Rozprzeglenie_Wozka";
      A(;
      O(;
      L     4;
      L     "DB_HMI_Wozek".HMI_OUT.Wartosc_Stosu_Elem_5;
      ==I;
      );
      O(;
      L     260;
      L     "DB_HMI_Wozek".HMI_OUT.Wartosc_Stosu_Elem_5;
      ==I;
      );
      );
      =     "Przejmij_z_I2";
NETWORK
TITLE =
//Przejmij palete ze stanowiska i3 (261!!!!!!!!!!!!!!!!)
      A     "DB_HMI_Wozek".HMI_IN.Wozek_W_Trybie_Auto;
      AN    "Foto_Wozek_Przod";
      AN    "Foto_Wozek_Tyl";
      A     "Rozprzeglenie_Wozka";
      A(;
      O(;
      L     5;
      L     "DB_HMI_Wozek".HMI_OUT.Wartosc_Stosu_Elem_5;
      ==I;
      );
      O(;
      L     261;
      L     "DB_HMI_Wozek".HMI_OUT.Wartosc_Stosu_Elem_5;
      ==I;
      );
      );
      =     "Przejmij_z_I3";
NETWORK
TITLE =
//Wartosc bufforu wozek
      L     "DB_HMI_Wozek".HMI_IN_OUT.Wartosc_Buforu_Wozek;
      T     "Wartosc_Bufforu_Help";
      NOP   0;
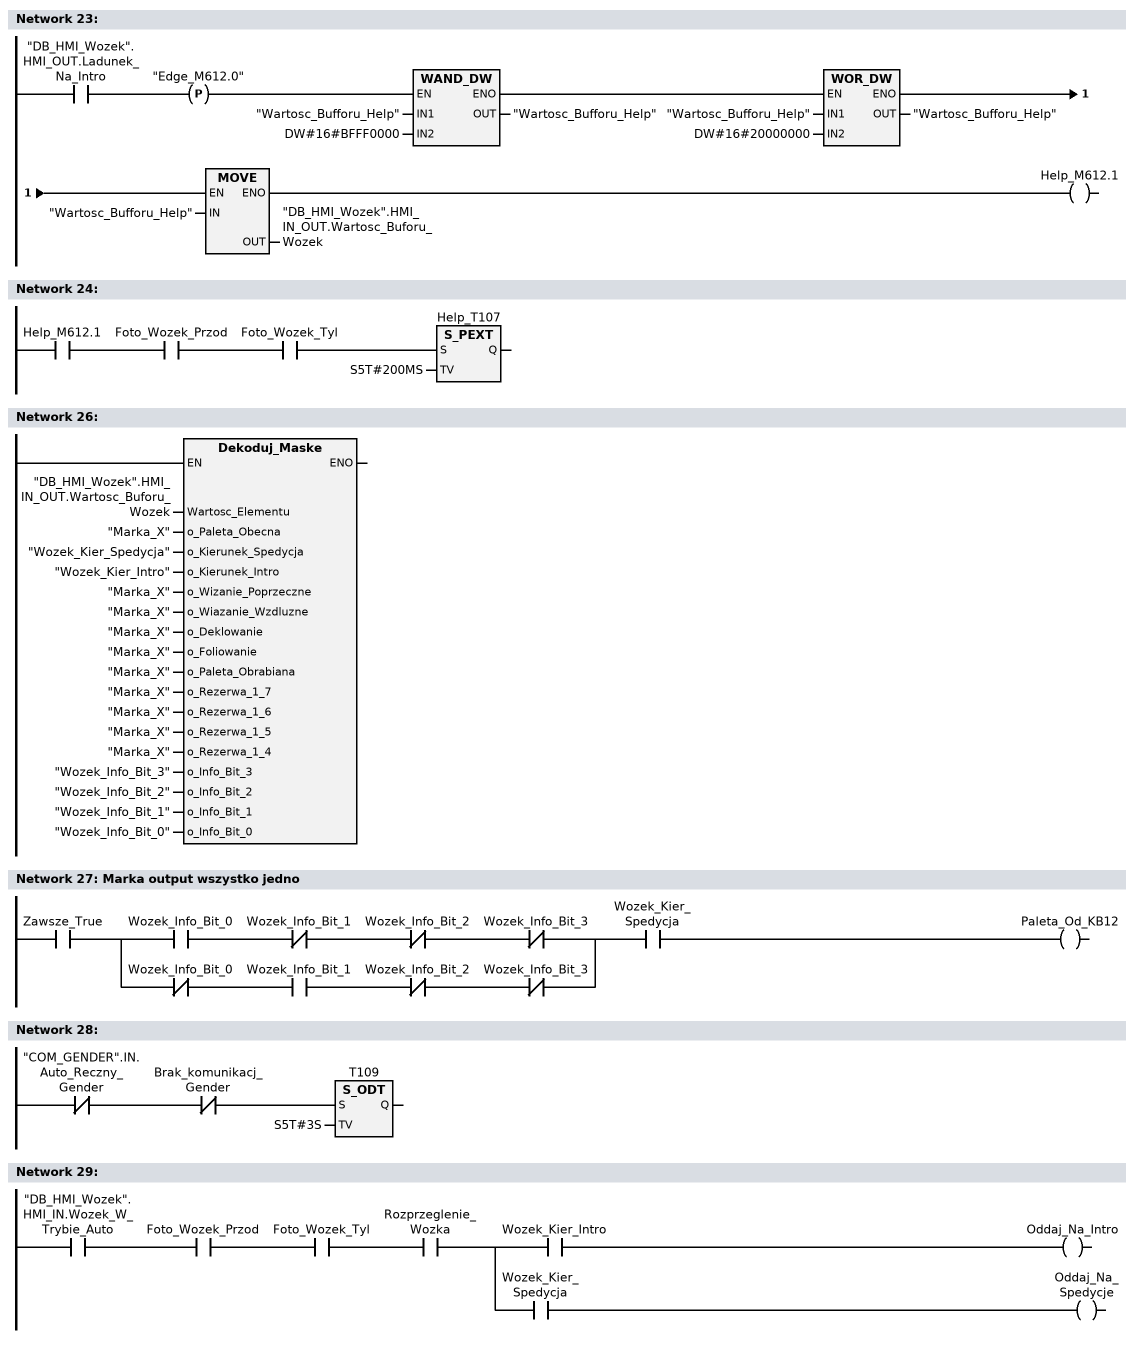
NETWORK
TITLE =
//Obsluga przycisku reset oddaj na intro
      A(;
      A(;
      A     "DB_HMI_Wozek".HMI_OUT.Ladunek_Na_Intro;
      FP    "Edge_M612.0";
      JNB   _009;
      L     "Wartosc_Bufforu_Help";
      L     DW#16#BFFF0000;
      AD;
      T     "Wartosc_Bufforu_Help";
      SET;
      SAVE;
      CLR;
_009: A     BR;
      );
      JNB   _00a;
      L     "Wartosc_Bufforu_Help";
      L     DW#16#20000000;
      OD;
      T     "Wartosc_Bufforu_Help";
      SET;
      SAVE;
      CLR;
_00a: A     BR;
      );
      JNB   _00b;
      L     "Wartosc_Bufforu_Help";
      T     "DB_HMI_Wozek".HMI_IN_OUT.Wartosc_Buforu_Wozek;
      SET;
      SAVE;
      CLR;
_00b: A     BR;
      =     "Help_M612.1";
NETWORK
TITLE =
//Ciag dalszy Reset palety gdy stoi pod genderm
//
      A     "Help_M612.1";
      A     "Foto_Wozek_Przod";
      A     "Foto_Wozek_Tyl";
      L     S5T#200MS;
      SE    "Help_T107";
      NOP   0;
      NOP   0;
      NOP   0;
      NOP   0;
NETWORK
TITLE =
NETWORK
TITLE =
//Dekoduj Wozek
//Marka x uzywana gdy elementy chwilowo niepotrzebne
      CALL  "Dekoduj_Maske" (
           Wartosc_Elementu         := "DB_HMI_Wozek".HMI_IN_OUT.Wartosc_Buforu_Wozek,
           o_Paleta_Obecna          := "Marka_X",
           o_Kierunek_Spedycja      := "Wozek_Kier_Spedycja",
           o_Kierunek_Intro         := "Wozek_Kier_Intro",
           o_Wizanie_Poprzeczne     := "Marka_X",
           o_Wiazanie_Wzdluzne      := "Marka_X",
           o_Deklowanie             := "Marka_X",
           o_Foliowanie             := "Marka_X",
           o_Paleta_Obrabiana       := "Marka_X",
           o_Rezerwa_1_7            := "Marka_X",
           o_Rezerwa_1_6            := "Marka_X",
           o_Rezerwa_1_5            := "Marka_X",
           o_Rezerwa_1_4            := "Marka_X",
           o_Info_Bit_3             := "Wozek_Info_Bit_3",
           o_Info_Bit_2             := "Wozek_Info_Bit_2",
           o_Info_Bit_1             := "Wozek_Info_Bit_1",
           o_Info_Bit_0             := "Wozek_Info_Bit_0");
NETWORK
TITLE = Marka output wszystko jedno
//Przesznuruj gdy gender zajety. Posc wtedy na bufory.Warunek IKEA
      A     "Zawsze_True";
      A(;
      A     "Wozek_Info_Bit_0";
      AN    "Wozek_Info_Bit_1";
      AN    "Wozek_Info_Bit_2";
      AN    "Wozek_Info_Bit_3";
      O;
      AN    "Wozek_Info_Bit_0";
      A     "Wozek_Info_Bit_1";
      AN    "Wozek_Info_Bit_2";
      AN    "Wozek_Info_Bit_3";
      );
      A     "Wozek_Kier_Spedycja";
      =     "Paleta_Od_KB12";
NETWORK
TITLE =
//Kiedy gender sie wywali w tryb reczny
      AN    "COM_GENDER".IN.Auto_Reczny_Gender;
      AN    "Brak_komunikacj_Gender";
      L     S5T#3S;
      SD    "T109";
      NOP   0;
      NOP   0;
      NOP   0;
      NOP   0;
NETWORK
TITLE =
//Oddaj palete na odpowiednie miejsce
      A     "DB_HMI_Wozek".HMI_IN.Wozek_W_Trybie_Auto;
      A     "Foto_Wozek_Przod";
      A     "Foto_Wozek_Tyl";
      A     "Rozprzeglenie_Wozka";
      =     L 0.0;
      A     L 0.0;
      A     "Wozek_Kier_Intro";
      =     "Oddaj_Na_Intro";
      A     L 0.0;
      A     "Wozek_Kier_Spedycja";
      =     "Oddaj_Na_Spedycje";
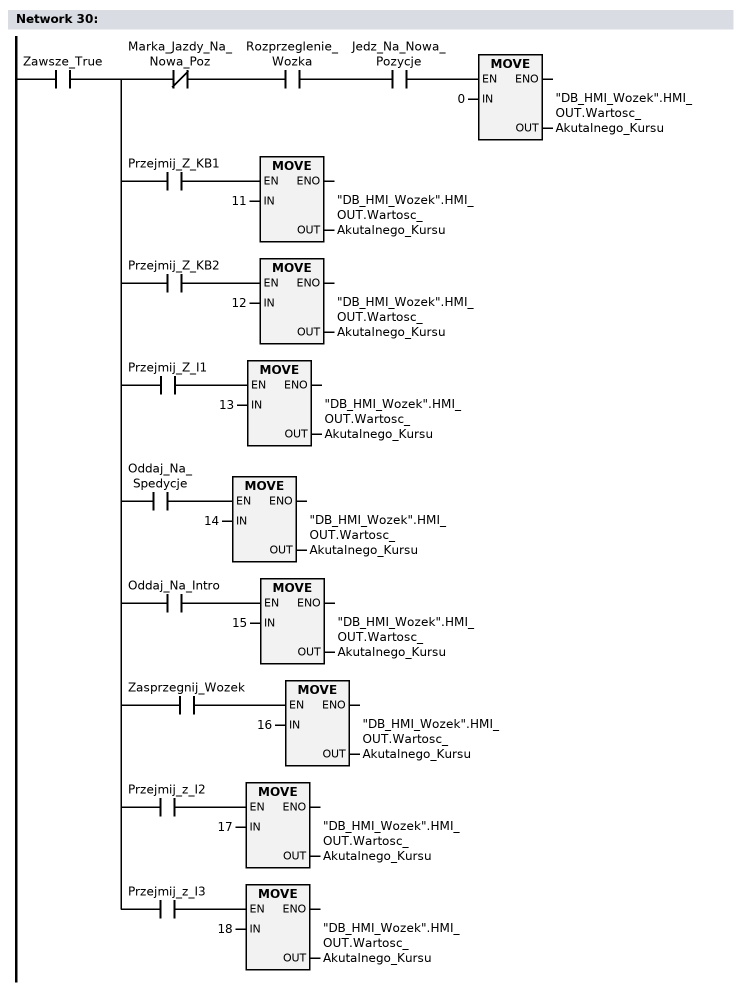
NETWORK
TITLE =
//Wyswietlenie gdzie jest jazda
//
//257 lub 1 -kb1  
//258 lub 2 -kb2
//259 lub 3 -buff
//11- kb1, 12kb2,  13-buff, 14-Gender, 15 Intro odbieranie, wozek zasprzeglony
      A     "Zawsze_True";
      =     L 0.0;
      A     L 0.0;
      AN    "Marka_Jazdy_Na_Nowa_Poz";
      A     "Rozprzeglenie_Wozka";
      A     "Jedz_Na_Nowa_Pozycje";
      JNB   _00c;
      L     0;
      T     "DB_HMI_Wozek".HMI_OUT.Wartosc_Akutalnego_Kursu;
_00c: NOP   0;
      A     L 0.0;
      A     "Przejmij_Z_KB1";
      JNB   _00d;
      L     11;
      T     "DB_HMI_Wozek".HMI_OUT.Wartosc_Akutalnego_Kursu;
_00d: NOP   0;
      A     L 0.0;
      A     "Przejmij_Z_KB2";
      JNB   _00e;
      L     12;
      T     "DB_HMI_Wozek".HMI_OUT.Wartosc_Akutalnego_Kursu;
_00e: NOP   0;
      A     L 0.0;
      A     "Przejmij_Z_I1";
      JNB   _00f;
      L     13;
      T     "DB_HMI_Wozek".HMI_OUT.Wartosc_Akutalnego_Kursu;
_00f: NOP   0;
      A     L 0.0;
      A     "Oddaj_Na_Spedycje";
      JNB   _010;
      L     14;
      T     "DB_HMI_Wozek".HMI_OUT.Wartosc_Akutalnego_Kursu;
_010: NOP   0;
      A     L 0.0;
      A     "Oddaj_Na_Intro";
      JNB   _011;
      L     15;
      T     "DB_HMI_Wozek".HMI_OUT.Wartosc_Akutalnego_Kursu;
_011: NOP   0;
      A     L 0.0;
      A     "Zasprzegnij_Wozek";
      JNB   _012;
      L     16;
      T     "DB_HMI_Wozek".HMI_OUT.Wartosc_Akutalnego_Kursu;
_012: NOP   0;
      A     L 0.0;
      A     "Przejmij_z_I2";
      JNB   _013;
      L     17;
      T     "DB_HMI_Wozek".HMI_OUT.Wartosc_Akutalnego_Kursu;
_013: NOP   0;
      A     L 0.0;
      A     "Przejmij_z_I3";
      JNB   _014;
      L     18;
      T     "DB_HMI_Wozek".HMI_OUT.Wartosc_Akutalnego_Kursu;
_014: NOP   0;
END_FUNCTION

FUNCTION "Send_Data" : VOID	// FC 700
//Funkcja Send_Data odpowiada za zapis duzej ilosci danych  z drugiego waskim 
//kanalem informacyjnym (kilku bajtowym). Funkcja 
//skonstruowana glownie do przesylu parametrow.
//
//Read_Data pracuje w parze z Share_Data
//
//Poszczegolne kroki w wysylaniu i odbieraniu
//
//i_Rozpocznij_Transmisje
//o_zadanie_transmisji     --> i_transmisja_ustanowiona
//ow_Nr_Bloku_Pobieranego  --> i_Blok_Pobierany_Zerezerwowany
//o_zadanie_danych         --> i_przesylanie_danych
//                         --> i_koniec_przesylania
//
//
//
//Po kazdej przeslanej danej musi dosjsc do inwersji bitu toggle
AUTHOR : Kng
NAME : COM
VERSION : 0.1
VAR_INPUT
  i_Reset : BOOL ;	//Reset Transmisji
  i_Rozpocznij_Transmisje : BOOL ;	//Wyslij dane (Wejscie aktywne na zbocze)
  i_Transmisja_Ustanowiona : BOOL ;	//Odpowiedz na zadanie transmisji
  i_Blok_Zew_Zarezerwowany : BOOL ;	//Potwierdzenie rezerwacji bloku w drugim urzadzeniu
  i_Przesylanie_Danych : BOOL ;	//Przesylanie w toku
  iw_Nr_Bloku_Nadpisu : INT ;	//Nr przesylanego bloku danych
  iw_Nr_Bloku_Poboru : INT ;	//Nr bloku gdzie dane sa zapisane
  iw_Ilosc_Max_Rekordow : INT ;	//Ilosc pobieranych rekordow
  iw_Rekord_Powracajacy : INT ;	//Potwierdzenie nr rekordu
END_VAR
VAR_OUTPUT
  o_Zadanie_Transmisji : BOOL ;	//Ustanowienie transmisji
  o_Zadanie_Danych : BOOL ;	//Zadanie wyslania indeksu danych
  o_Koniec_Nadawania : BOOL ;	//Sygnal opadajacy
  ow_Nr_Bloku_Nadpisu : INT ;
  ow_Nr_Rekordu : INT ;
  ow_Kanal_Nadawania : INT ;	//Kanal wysylania
END_VAR
VAR_IN_OUT
  io_Help_Word : WORD ;
  iow_NR_Petli : INT ;	//Nr petli danych
END_VAR
VAR_TEMP
  Przesylanie_Aktywne : BOOL ;
  L_Rozpocznij_Transfer : BOOL ;
  Zbocze_1 : BOOL ;
  Temp_Byte : BYTE ;
  Help_Word_2 : WORD ;
  L_NR_Bloku_Zapisu : WORD ;
  L_Nr_Recordu : DWORD ;
  L_DW_Licznik_Rekordow : DWORD ;
END_VAR
BEGIN
NETWORK
TITLE =
//Ten Network celowo jest wolny
NETWORK
TITLE =
//Pobranie zmiennych pomocniczych
      L     #io_Help_Word;
      T     LW 0;
NETWORK
TITLE =
//Pobierz nazwe bloku kopiowanego
      L     #iw_Nr_Bloku_Poboru;	// Nr bloku db
      T     #L_NR_Bloku_Zapisu;
      OPN   DB [#L_NR_Bloku_Zapisu];	// Otwarcie db
NETWORK
TITLE =
//Rzadanie transmisji
//
      A     #i_Rozpocznij_Transmisje;
      FP    #Zbocze_1;
      S     #L_Rozpocznij_Transfer;
      S     #o_Koniec_Nadawania;
      JCN   zer;
      L     0;
      T     #iow_NR_Petli;
zer:  NOP   0;
      A     #L_Rozpocznij_Transfer;
      =     #o_Zadanie_Transmisji;
NETWORK
TITLE =
//Przeslanie nazwy bloku 
//Przeslanie nazwy bloku odbierania danych. Potwierdzeni wraca bitem
//blok_Odb_Zarezerwowany
      A     #L_Rozpocznij_Transfer;
      A     #i_Transmisja_Ustanowiona;
      JCN   et_1;
      L     #iw_Nr_Bloku_Nadpisu;
      T     #ow_Nr_Bloku_Nadpisu;
      JU    et_2;
et_1: NOP   0;
      L     0;
      T     #ow_Nr_Bloku_Nadpisu;
et_2: NOP   0;
NETWORK
TITLE =
//Przeslanie Pierwszego podwojenego slowa w celu nawiazania komunikacji
      A     #L_Rozpocznij_Transfer;
      A     #i_Blok_Zew_Zarezerwowany;
      A     #i_Transmisja_Ustanowiona;
      =     #o_Zadanie_Danych;
NETWORK
TITLE =
//Otrzymanie potwierdzenia
      A     #L_Rozpocznij_Transfer;
      A     #i_Blok_Zew_Zarezerwowany;
      A     #i_Transmisja_Ustanowiona;
      A     #i_Przesylanie_Danych;
      =     #Przesylanie_Aktywne;
//Wylicz nr rekordu
      L     #iow_NR_Petli;
      L     2;
      *I;
      ITD;
      SLD   3;
      T     #L_DW_Licznik_Rekordow;
      L     #iow_NR_Petli;
      T     #ow_Nr_Rekordu;
// podlicz rekordy
      A(;
      L     #iow_NR_Petli;
      L     #iw_Rekord_Powracajacy;
      ==I;
      );
      A     #Przesylanie_Aktywne;
      JCN   et_3;
      L     DBW [#L_DW_Licznik_Rekordow];	//h
      T     #ow_Kanal_Nadawania;
      L     #iow_NR_Petli;
      L     1;
      +I;
      T     #iow_NR_Petli;
et_3: NOP   0;
//Zakoncz gdy koniec iteracji
      O(;
      L     #iow_NR_Petli;
      L     #iw_Ilosc_Max_Rekordow;
      >=I;
      );
      O     #i_Reset;
      JCN   d0;
      L     0;
      T     #iw_Ilosc_Max_Rekordow;
      SET;
      R     #L_Rozpocznij_Transfer;
      R     #o_Koniec_Nadawania;
d0:   NOP   0;
NETWORK
TITLE =
//Zapis bitow przejsciowych
      L     LW 0;
      T     #io_Help_Word;
END_FUNCTION

FUNCTION "Read_Data" : VOID	// FC 702
//Funkcja Read_Data odpowiada za odczyt duzej ilosci danych  z drugiego waskim 
//kanalem informacyjnym (kilku bajtowym). Funkcja 
//skonstruowana glownie do przesylu parametrow.
//
//Read_Data pracuje w parze z Share_Data
//
//Poszczegolne kroki w wysylaniu i odbieraniu
//
//i_Rozpocznij_Transmisje
//o_zadanie_transmisji     --> i_transmisja_ustanowiona
//ow_Nr_Bloku_Pobieranego  --> i_Blok_Pobierany_Zerezerwowany
//o_zadanie_danych         --> i_przesylanie_danych
//                         --> i_koniec_przesylania
//
//
//
//Po kazdej przeslanej danej musi dosjsc do inwersji bitu toggle
AUTHOR : Kng
NAME : COM
VERSION : 0.1
VAR_INPUT
  i_Reset : BOOL ;	//Reset Transmisji
  i_Rozpocznij_Transmisje : BOOL ;	//Wyslij dane (Wejscie aktywne na zbocze)
  i_Transmisja_Ustanowiona : BOOL ;	//Odpowiedz na zadanie transmisji
  i_Blok_Zew_Zarezerwowany : BOOL ;	//Potwierdzenie rezerwacji bloku w drugim urzadzeniu
  i_Przesylanie_Danych : BOOL ;	//Przesylanie w toku
  iw_Nr_Bloku_Pobieranego : INT ;	//Nr przesylanego bloku danych
  iw_Nr_Bloku_Zapisu : INT ;	//Nr bloku gdzie dane sa zapisane
  iw_Kanal_Odbierania : INT ;	//Kanal danych pobieranych
  iw_Ilosc_Max_Rekordow : INT ;	//Ilosc pobieranych rekordow
  iw_Rekord_Powracajacy : INT ;	//Potwierdzenie nr rekordu
END_VAR
VAR_OUTPUT
  o_Zadanie_Transmisji : BOOL ;	//Ustanowienie transmisji
  o_Zadanie_Danych : BOOL ;	//Zadanie wyslania indeksu danych
  o_Koniec_Nadawania : BOOL ;	//Sygnal opadajacy
  ow_Nr_Bloku_Pobieranego : INT ;
  ow_Nr_Rekordu : INT ;
END_VAR
VAR_IN_OUT
  io_Help_Word : WORD ;
  iow_NR_Petli : INT ;	//Nr petli danych
END_VAR
VAR_TEMP
  Przesylanie_Aktywne : BOOL ;
  L_Rozpocznij_Transfer : BOOL ;
  Zbocze_1 : BOOL ;
  Temp_Byte : BYTE ;
  Help_Word_2 : WORD ;
  L_NR_Bloku_Zapisu : WORD ;
  L_Nr_Recordu : DWORD ;
  L_DW_Licznik_Rekordow : DWORD ;
END_VAR
BEGIN
NETWORK
TITLE =
//Ten Network celowo jest wolny
NETWORK
TITLE =
//Pobranie zmiennych pomocniczych
      L     #io_Help_Word;
      T     LW 0;
NETWORK
TITLE =
//Pobierz nazwe bloku kopiowanego
      L     #iw_Nr_Bloku_Zapisu;	// Nr bloku db
      T     #L_NR_Bloku_Zapisu;
      OPN   DB [#L_NR_Bloku_Zapisu];	// Otwarcie db
NETWORK
TITLE =
//Rzadanie transmisji
//
      A     #i_Rozpocznij_Transmisje;
      FP    #Zbocze_1;
      S     #L_Rozpocznij_Transfer;
      S     #o_Koniec_Nadawania;
      JCN   zer;
      L     0;
      T     #iow_NR_Petli;
zer:  NOP   0;
      A     #L_Rozpocznij_Transfer;
      =     #o_Zadanie_Transmisji;
NETWORK
TITLE =
//Przeslanie nazwy bloku 
//Przeslanie nazwy bloku odbierania danych. Potwierdzeni wraca bitem
//blok_Odb_Zarezerwowany
      A     #L_Rozpocznij_Transfer;
      A     #i_Transmisja_Ustanowiona;
      JCN   et_1;
      L     #iw_Nr_Bloku_Pobieranego;
      T     #ow_Nr_Bloku_Pobieranego;
      JU    et_2;
et_1: NOP   0;
      L     0;
      T     #ow_Nr_Bloku_Pobieranego;
et_2: NOP   0;
NETWORK
TITLE =
//Przeslanie Pierwszego podwojenego slowa w celu nawiazania komunikacji
      A     #L_Rozpocznij_Transfer;
      A     #i_Blok_Zew_Zarezerwowany;
      A     #i_Transmisja_Ustanowiona;
      =     #o_Zadanie_Danych;
NETWORK
TITLE =
//Otrzymanie potwierdzenia
      A     #L_Rozpocznij_Transfer;
      A     #i_Blok_Zew_Zarezerwowany;
      A     #i_Transmisja_Ustanowiona;
      A     #i_Przesylanie_Danych;
      =     #Przesylanie_Aktywne;
//Wylicz nr rekordu
      L     #iow_NR_Petli;
      L     2;
      *I;
      ITD;
      SLD   3;
      T     #L_DW_Licznik_Rekordow;
      L     #iow_NR_Petli;
      T     #ow_Nr_Rekordu;
// podlicz rekordy
      A(;
      L     #iow_NR_Petli;
      L     #iw_Rekord_Powracajacy;
      ==I;
      );
      A     #Przesylanie_Aktywne;
      JCN   et_3;
      L     #iw_Kanal_Odbierania;
      T     DBW [#L_DW_Licznik_Rekordow];	//Zapisanie danych
      L     #iow_NR_Petli;
      L     1;
      +I;
      T     #iow_NR_Petli;
et_3: NOP   0;
//Zakoncz gdy koniec iteracji
      O(;
      L     #iow_NR_Petli;
      L     #iw_Ilosc_Max_Rekordow;
      >=I;
      );
      O     #i_Reset;
      JCN   d0;
      L     0;
      T     #iw_Ilosc_Max_Rekordow;
      SET;
      R     #L_Rozpocznij_Transfer;
      R     #o_Koniec_Nadawania;
d0:   NOP   0;
NETWORK
TITLE =
//Zapis bitow przejsciowych
      L     LW 0;
      T     #io_Help_Word;
END_FUNCTION

FUNCTION "Ekran_Para_Wozek" : VOID	// FC 1701
VERSION : 0.1
VAR_INPUT
  Ekran_Aktywny : BOOL ;
  Timmer_Opoz : TIMER ;
END_VAR
VAR_OUTPUT
  Aktywne_Read : BOOL ;
  Aktywne_Write : BOOL ;
  Aktywna_Funkcja : BOOL ;
END_VAR
BEGIN
NETWORK
TITLE =
//Ten network celowo jest wolny
//inputy to i160
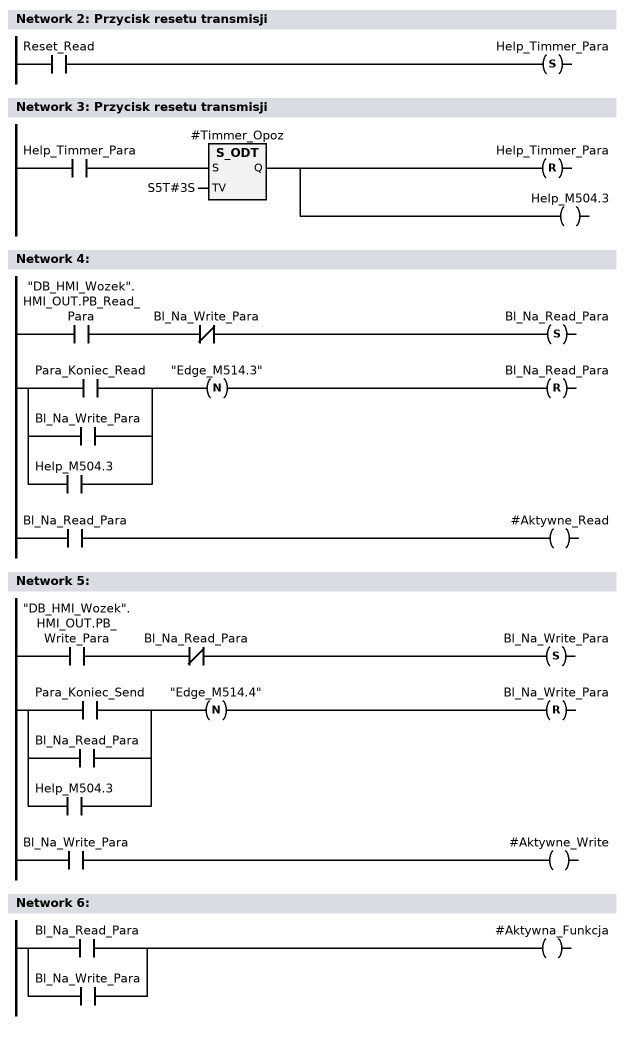
NETWORK
TITLE = Przycisk resetu transmisji
      A     "Reset_Read";
      S     "Help_Timmer_Para";
NETWORK
TITLE = Przycisk resetu transmisji
      A     "Help_Timmer_Para";
      L     S5T#3S;
      SD    #Timmer_Opoz;
      NOP   0;
      NOP   0;
      NOP   0;
      A     #Timmer_Opoz;
      R     "Help_Timmer_Para";
      =     "Help_M504.3";
NETWORK
TITLE =
//Blokada NA Read
      A     "DB_HMI_Wozek".HMI_OUT.PB_Read_Para;
      AN    "Bl_Na_Write_Para";
      S     "Bl_Na_Read_Para";
      A(;
      O     "Para_Koniec_Read";
      O     "Bl_Na_Write_Para";
      O     "Help_M504.3";
      );
      FN    "Edge_M514.3";
      R     "Bl_Na_Read_Para";
      A     "Bl_Na_Read_Para";
      =     #Aktywne_Read;
NETWORK
TITLE =
//Blokada NA write
      A     "DB_HMI_Wozek".HMI_OUT.PB_Write_Para;
      AN    "Bl_Na_Read_Para";
      S     "Bl_Na_Write_Para";
      A(;
      O     "Para_Koniec_Send";
      O     "Bl_Na_Read_Para";
      O     "Help_M504.3";
      );
      FN    "Edge_M514.4";
      R     "Bl_Na_Write_Para";
      A     "Bl_Na_Write_Para";
      =     #Aktywne_Write;
NETWORK
TITLE =
      O     "Bl_Na_Read_Para";
      O     "Bl_Na_Write_Para";
      =     #Aktywna_Funkcja;
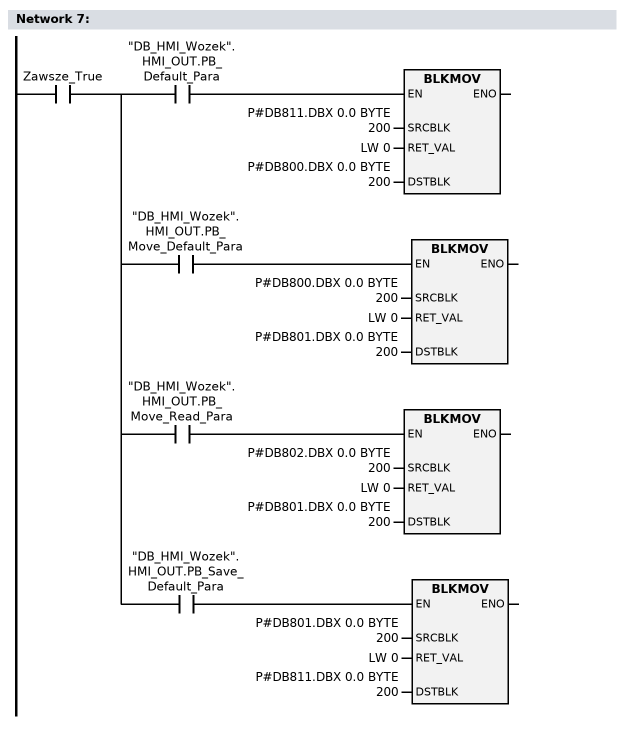
NETWORK
TITLE =
      A     "Zawsze_True";
      =     L 2.0;
      A     L 2.0;
      A     "DB_HMI_Wozek".HMI_OUT.PB_Default_Para;
      JNB   _001;
      CALL  "BLKMOV" (
           SRCBLK                   := P#DB811.DBX 0.0 BYTE 200,
           RET_VAL                  := LW 0,
           DSTBLK                   := P#DB800.DBX 0.0 BYTE 200);
_001: NOP   0;
      A     L 2.0;
      A     "DB_HMI_Wozek".HMI_OUT.PB_Move_Default_Para;
      JNB   _002;
      CALL  "BLKMOV" (
           SRCBLK                   := P#DB800.DBX 0.0 BYTE 200,
           RET_VAL                  := LW 0,
           DSTBLK                   := P#DB801.DBX 0.0 BYTE 200);
_002: NOP   0;
      A     L 2.0;
      A     "DB_HMI_Wozek".HMI_OUT.PB_Move_Read_Para;
      JNB   _003;
      CALL  "BLKMOV" (
           SRCBLK                   := P#DB802.DBX 0.0 BYTE 200,
           RET_VAL                  := LW 0,
           DSTBLK                   := P#DB801.DBX 0.0 BYTE 200);
_003: NOP   0;
      A     L 2.0;
      A     "DB_HMI_Wozek".HMI_OUT.PB_Save_Default_Para;
      JNB   _004;
      CALL  "BLKMOV" (
           SRCBLK                   := P#DB801.DBX 0.0 BYTE 200,
           RET_VAL                  := LW 0,
           DSTBLK                   := P#DB811.DBX 0.0 BYTE 200);
_004: NOP   0;
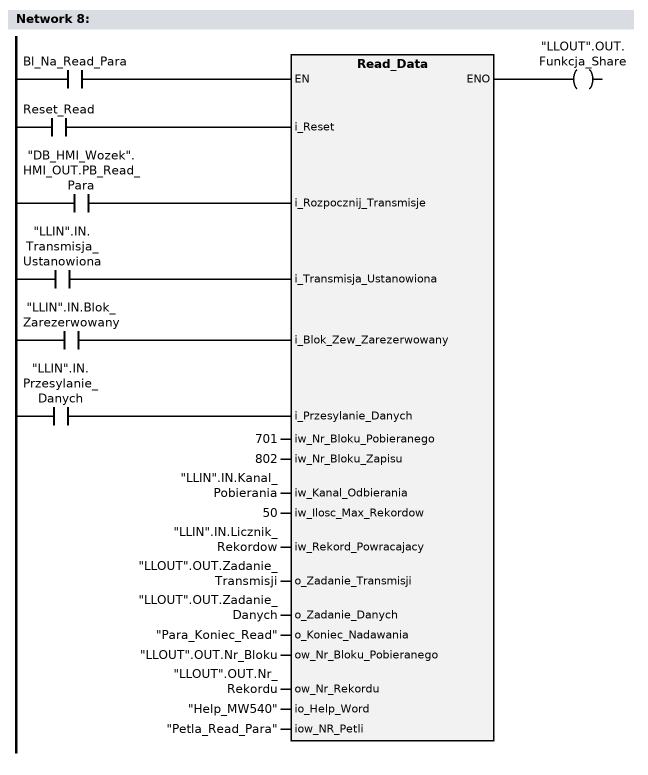
NETWORK
TITLE =
//Funkcja poboru danych
//
      A     "Reset_Read";
      =     L 2.0;
      BLD   103;
      A     "DB_HMI_Wozek".HMI_OUT.PB_Read_Para;
      =     L 2.1;
      BLD   103;
      A     "LLIN".IN.Transmisja_Ustanowiona;
      =     L 2.2;
      BLD   103;
      A     "LLIN".IN.Blok_Zarezerwowany;
      =     L 2.3;
      BLD   103;
      A     "LLIN".IN.Przesylanie_Danych;
      =     L 2.4;
      BLD   103;
      A     "Bl_Na_Read_Para";
      JNB   _005;
      CALL  "Read_Data" (
           i_Reset                  := L 2.0,
           i_Rozpocznij_Transmisje  := L 2.1,
           i_Transmisja_Ustanowiona := L 2.2,
           i_Blok_Zew_Zarezerwowany := L 2.3,
           i_Przesylanie_Danych     := L 2.4,
           iw_Nr_Bloku_Pobieranego  := 701,
           iw_Nr_Bloku_Zapisu       := 802,
           iw_Kanal_Odbierania      := "LLIN".IN.Kanal_Pobierania,
           iw_Ilosc_Max_Rekordow    := 50,
           iw_Rekord_Powracajacy    := "LLIN".IN.Licznik_Rekordow,
           o_Zadanie_Transmisji     := "LLOUT".OUT.Zadanie_Transmisji,
           o_Zadanie_Danych         := "LLOUT".OUT.Zadanie_Danych,
           o_Koniec_Nadawania       := "Para_Koniec_Read",
           ow_Nr_Bloku_Pobieranego  := "LLOUT".OUT.Nr_Bloku,
           ow_Nr_Rekordu            := "LLOUT".OUT.Nr_Rekordu,
           io_Help_Word             := "Help_MW540",
           iow_NR_Petli             := "Petla_Read_Para");
_005: A     BR;
      =     "LLOUT".OUT.Funkcja_Share;
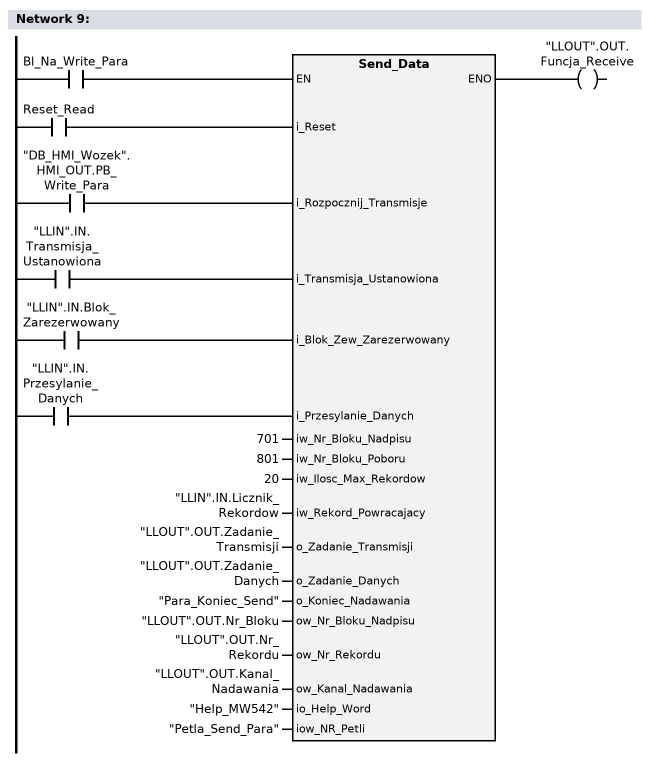
NETWORK
TITLE =
      A     "Reset_Read";
      =     L 2.0;
      BLD   103;
      A     "DB_HMI_Wozek".HMI_OUT.PB_Write_Para;
      =     L 2.1;
      BLD   103;
      A     "LLIN".IN.Transmisja_Ustanowiona;
      =     L 2.2;
      BLD   103;
      A     "LLIN".IN.Blok_Zarezerwowany;
      =     L 2.3;
      BLD   103;
      A     "LLIN".IN.Przesylanie_Danych;
      =     L 2.4;
      BLD   103;
      A     "Bl_Na_Write_Para";
      JNB   _006;
      CALL  "Send_Data" (
           i_Reset                  := L 2.0,
           i_Rozpocznij_Transmisje  := L 2.1,
           i_Transmisja_Ustanowiona := L 2.2,
           i_Blok_Zew_Zarezerwowany := L 2.3,
           i_Przesylanie_Danych     := L 2.4,
           iw_Nr_Bloku_Nadpisu      := 701,
           iw_Nr_Bloku_Poboru       := 801,
           iw_Ilosc_Max_Rekordow    := 20,
           iw_Rekord_Powracajacy    := "LLIN".IN.Licznik_Rekordow,
           o_Zadanie_Transmisji     := "LLOUT".OUT.Zadanie_Transmisji,
           o_Zadanie_Danych         := "LLOUT".OUT.Zadanie_Danych,
           o_Koniec_Nadawania       := "Para_Koniec_Send",
           ow_Nr_Bloku_Nadpisu      := "LLOUT".OUT.Nr_Bloku,
           ow_Nr_Rekordu            := "LLOUT".OUT.Nr_Rekordu,
           ow_Kanal_Nadawania       := "LLOUT".OUT.Kanal_Nadawania,
           io_Help_Word             := "Help_MW542",
           iow_NR_Petli             := "Petla_Send_Para");
_006: A     BR;
      =     "LLOUT".OUT.Funcja_Receive;
END_FUNCTION

FUNCTION "Ekran_Kier_KB1" : VOID	// FC 1720
VERSION : 0.1
VAR_INPUT
  Ekran_Aktywny : BOOL ;
  Timmer_Opoz : TIMER ;
END_VAR
VAR_OUTPUT
  Aktywne_Read : BOOL ;
  Aktywne_Write : BOOL ;
  Aktywna_Funkcja : BOOL ;
END_VAR
BEGIN
NETWORK
TITLE =
//Ten network celowo jest wolny
//inputy to i160
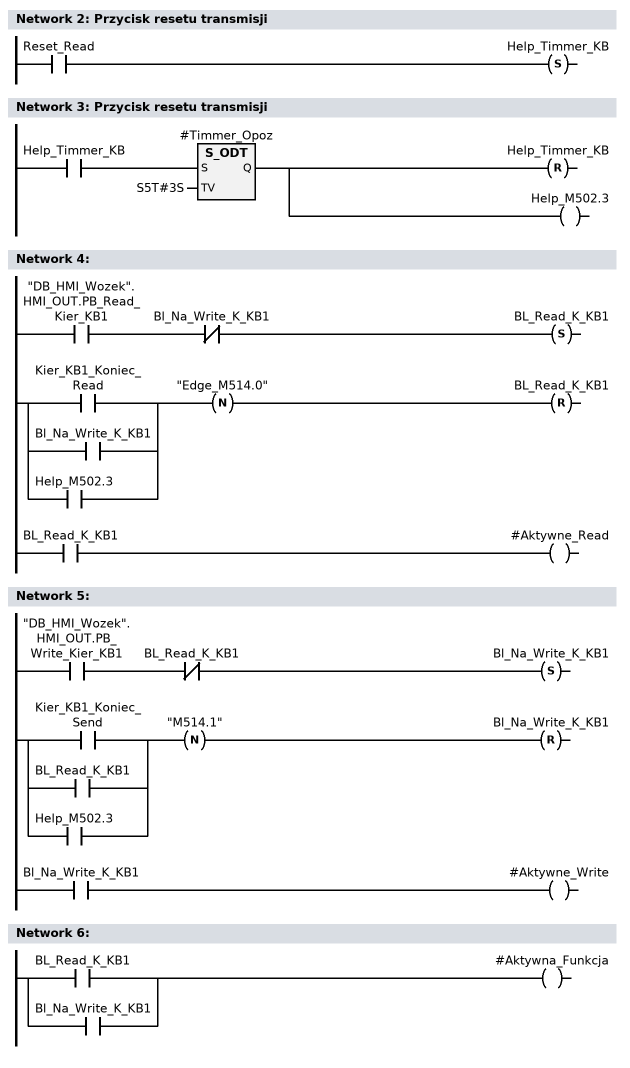
NETWORK
TITLE = Przycisk resetu transmisji
      A     "Reset_Read";
      S     "Help_Timmer_KB";
NETWORK
TITLE = Przycisk resetu transmisji
      A     "Help_Timmer_KB";
      L     S5T#3S;
      SD    #Timmer_Opoz;
      NOP   0;
      NOP   0;
      NOP   0;
      A     #Timmer_Opoz;
      R     "Help_Timmer_KB";
      =     "Help_M502.3";
NETWORK
TITLE =
//Blokada NA Read
      A     "DB_HMI_Wozek".HMI_OUT.PB_Read_Kier_KB1;
      AN    "Bl_Na_Write_K_KB1";
      S     "BL_Read_K_KB1";
      A(;
      O     "Kier_KB1_Koniec_Read";
      O     "Bl_Na_Write_K_KB1";
      O     "Help_M502.3";
      );
      FN    "Edge_M514.0";
      R     "BL_Read_K_KB1";
      A     "BL_Read_K_KB1";
      =     #Aktywne_Read;
NETWORK
TITLE =
//Blokada NA write
      A     "DB_HMI_Wozek".HMI_OUT.PB_Write_Kier_KB1;
      AN    "BL_Read_K_KB1";
      S     "Bl_Na_Write_K_KB1";
      A(;
      O     "Kier_KB1_Koniec_Send";
      O     "BL_Read_K_KB1";
      O     "Help_M502.3";
      );
      FN    "M514.1";
      R     "Bl_Na_Write_K_KB1";
      A     "Bl_Na_Write_K_KB1";
      =     #Aktywne_Write;
NETWORK
TITLE =
      O     "BL_Read_K_KB1";
      O     "Bl_Na_Write_K_KB1";
      =     #Aktywna_Funkcja;
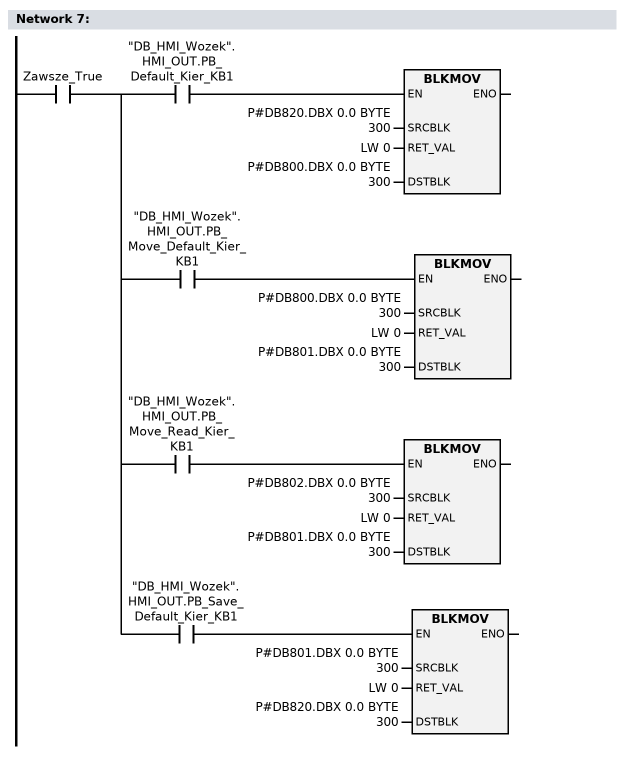
NETWORK
TITLE =
      A     "Zawsze_True";
      =     L 2.0;
      A     L 2.0;
      A     "DB_HMI_Wozek".HMI_OUT.PB_Default_Kier_KB1;
      JNB   _001;
      CALL  "BLKMOV" (
           SRCBLK                   := P#DB820.DBX 0.0 BYTE 300,
           RET_VAL                  := LW 0,
           DSTBLK                   := P#DB800.DBX 0.0 BYTE 300);
_001: NOP   0;
      A     L 2.0;
      A     "DB_HMI_Wozek".HMI_OUT.PB_Move_Default_Kier_KB1;
      JNB   _002;
      CALL  "BLKMOV" (
           SRCBLK                   := P#DB800.DBX 0.0 BYTE 300,
           RET_VAL                  := LW 0,
           DSTBLK                   := P#DB801.DBX 0.0 BYTE 300);
_002: NOP   0;
      A     L 2.0;
      A     "DB_HMI_Wozek".HMI_OUT.PB_Move_Read_Kier_KB1;
      JNB   _003;
      CALL  "BLKMOV" (
           SRCBLK                   := P#DB802.DBX 0.0 BYTE 300,
           RET_VAL                  := LW 0,
           DSTBLK                   := P#DB801.DBX 0.0 BYTE 300);
_003: NOP   0;
      A     L 2.0;
      A     "DB_HMI_Wozek".HMI_OUT.PB_Save_Default_Kier_KB1;
      JNB   _004;
      CALL  "BLKMOV" (
           SRCBLK                   := P#DB801.DBX 0.0 BYTE 300,
           RET_VAL                  := LW 0,
           DSTBLK                   := P#DB820.DBX 0.0 BYTE 300);
_004: NOP   0;
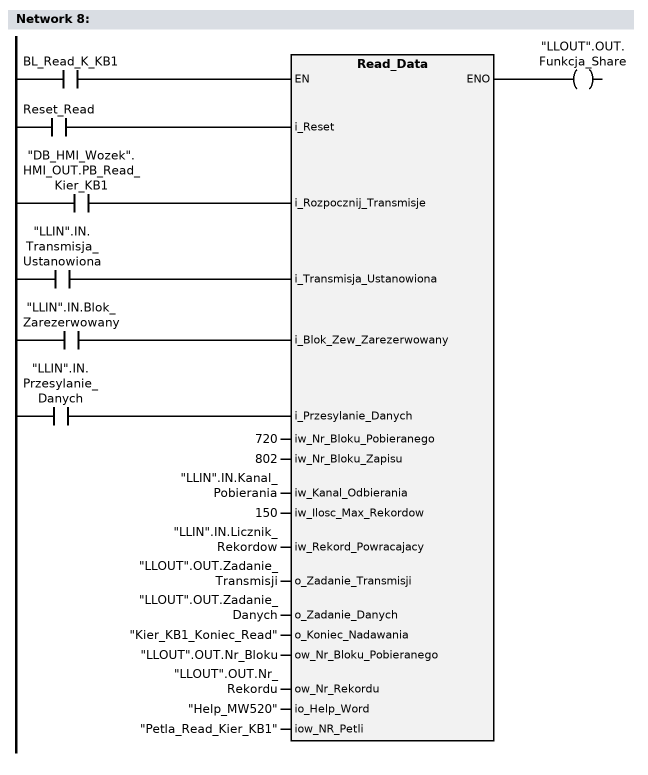
NETWORK
TITLE =
//Funkcja poboru danych
//
      A     "Reset_Read";
      =     L 2.0;
      BLD   103;
      A     "DB_HMI_Wozek".HMI_OUT.PB_Read_Kier_KB1;
      =     L 2.1;
      BLD   103;
      A     "LLIN".IN.Transmisja_Ustanowiona;
      =     L 2.2;
      BLD   103;
      A     "LLIN".IN.Blok_Zarezerwowany;
      =     L 2.3;
      BLD   103;
      A     "LLIN".IN.Przesylanie_Danych;
      =     L 2.4;
      BLD   103;
      A     "BL_Read_K_KB1";
      JNB   _005;
      CALL  "Read_Data" (
           i_Reset                  := L 2.0,
           i_Rozpocznij_Transmisje  := L 2.1,
           i_Transmisja_Ustanowiona := L 2.2,
           i_Blok_Zew_Zarezerwowany := L 2.3,
           i_Przesylanie_Danych     := L 2.4,
           iw_Nr_Bloku_Pobieranego  := 720,
           iw_Nr_Bloku_Zapisu       := 802,
           iw_Kanal_Odbierania      := "LLIN".IN.Kanal_Pobierania,
           iw_Ilosc_Max_Rekordow    := 150,
           iw_Rekord_Powracajacy    := "LLIN".IN.Licznik_Rekordow,
           o_Zadanie_Transmisji     := "LLOUT".OUT.Zadanie_Transmisji,
           o_Zadanie_Danych         := "LLOUT".OUT.Zadanie_Danych,
           o_Koniec_Nadawania       := "Kier_KB1_Koniec_Read",
           ow_Nr_Bloku_Pobieranego  := "LLOUT".OUT.Nr_Bloku,
           ow_Nr_Rekordu            := "LLOUT".OUT.Nr_Rekordu,
           io_Help_Word             := "Help_MW520",
           iow_NR_Petli             := "Petla_Read_Kier_KB1");
_005: A     BR;
      =     "LLOUT".OUT.Funkcja_Share;
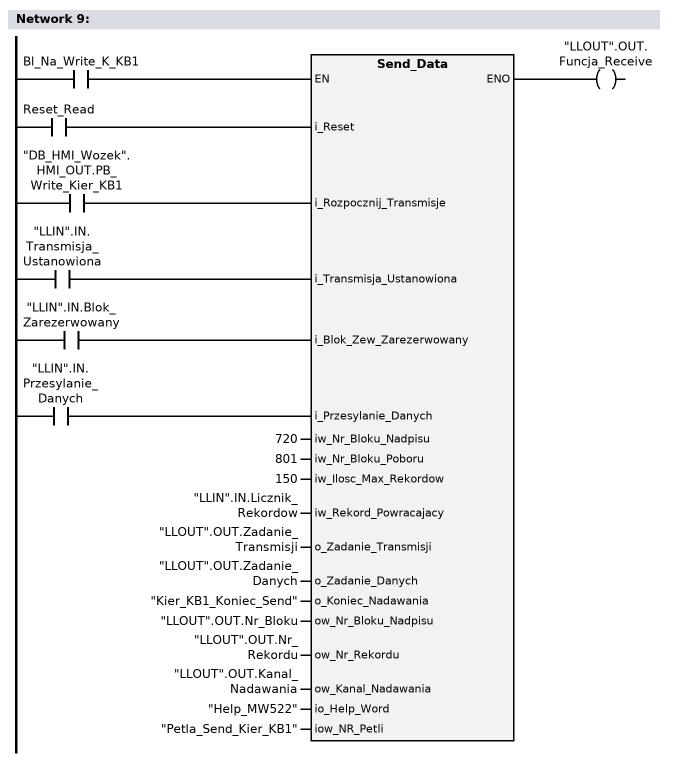
NETWORK
TITLE =
      A     "Reset_Read";
      =     L 2.0;
      BLD   103;
      A     "DB_HMI_Wozek".HMI_OUT.PB_Write_Kier_KB1;
      =     L 2.1;
      BLD   103;
      A     "LLIN".IN.Transmisja_Ustanowiona;
      =     L 2.2;
      BLD   103;
      A     "LLIN".IN.Blok_Zarezerwowany;
      =     L 2.3;
      BLD   103;
      A     "LLIN".IN.Przesylanie_Danych;
      =     L 2.4;
      BLD   103;
      A     "Bl_Na_Write_K_KB1";
      JNB   _006;
      CALL  "Send_Data" (
           i_Reset                  := L 2.0,
           i_Rozpocznij_Transmisje  := L 2.1,
           i_Transmisja_Ustanowiona := L 2.2,
           i_Blok_Zew_Zarezerwowany := L 2.3,
           i_Przesylanie_Danych     := L 2.4,
           iw_Nr_Bloku_Nadpisu      := 720,
           iw_Nr_Bloku_Poboru       := 801,
           iw_Ilosc_Max_Rekordow    := 150,
           iw_Rekord_Powracajacy    := "LLIN".IN.Licznik_Rekordow,
           o_Zadanie_Transmisji     := "LLOUT".OUT.Zadanie_Transmisji,
           o_Zadanie_Danych         := "LLOUT".OUT.Zadanie_Danych,
           o_Koniec_Nadawania       := "Kier_KB1_Koniec_Send",
           ow_Nr_Bloku_Nadpisu      := "LLOUT".OUT.Nr_Bloku,
           ow_Nr_Rekordu            := "LLOUT".OUT.Nr_Rekordu,
           ow_Kanal_Nadawania       := "LLOUT".OUT.Kanal_Nadawania,
           io_Help_Word             := "Help_MW522",
           iow_NR_Petli             := "Petla_Send_Kier_KB1");
_006: A     BR;
      =     "LLOUT".OUT.Funcja_Receive;
END_FUNCTION

FUNCTION "Ekran_Kier_Rot" : VOID	// FC 1721
VERSION : 0.1
VAR_INPUT
  Ekran_Aktywny : BOOL ;
  Timmer_Opoz : TIMER ;
END_VAR
VAR_OUTPUT
  Aktywne_Read : BOOL ;
  Aktywne_Write : BOOL ;
  Aktywna_Funkcja : BOOL ;
END_VAR
BEGIN
NETWORK
TITLE =
//Ten network celowo jest wolny
//inputy to i160
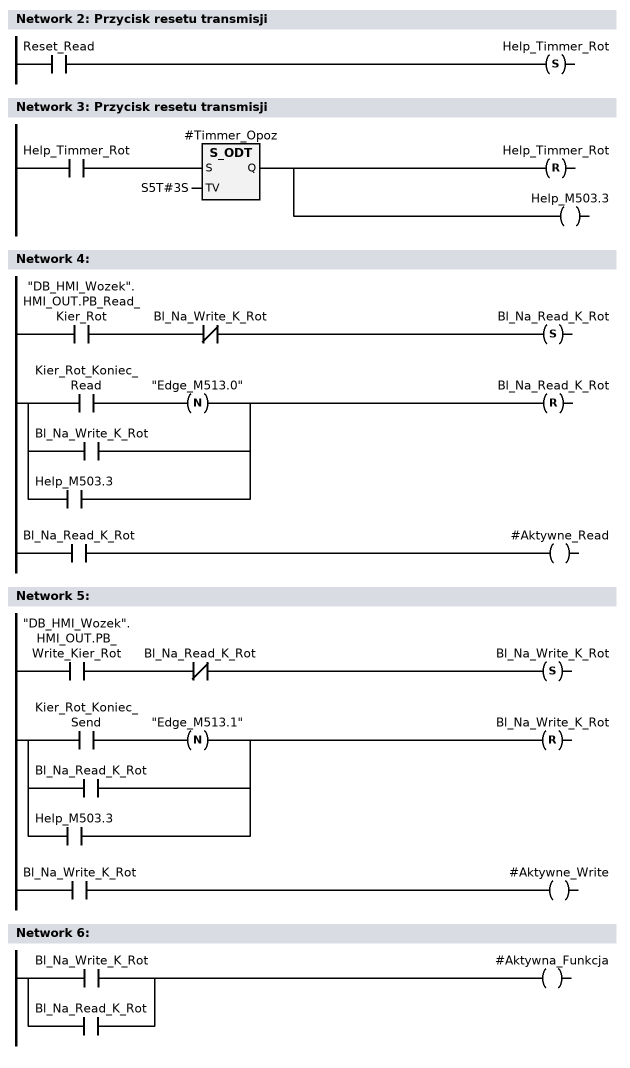
NETWORK
TITLE = Przycisk resetu transmisji
      A     "Reset_Read";
      S     "Help_Timmer_Rot";
NETWORK
TITLE = Przycisk resetu transmisji
      A     "Help_Timmer_Rot";
      L     S5T#3S;
      SD    #Timmer_Opoz;
      NOP   0;
      NOP   0;
      NOP   0;
      A     #Timmer_Opoz;
      R     "Help_Timmer_Rot";
      =     "Help_M503.3";
NETWORK
TITLE =
//Blokada NA Read
      A     "DB_HMI_Wozek".HMI_OUT.PB_Read_Kier_Rot;
      AN    "Bl_Na_Write_K_Rot";
      S     "Bl_Na_Read_K_Rot";
      A(;
      A     "Kier_Rot_Koniec_Read";
      FN    "Edge_M513.0";
      O     "Bl_Na_Write_K_Rot";
      O     "Help_M503.3";
      );
      R     "Bl_Na_Read_K_Rot";
      A     "Bl_Na_Read_K_Rot";
      =     #Aktywne_Read;
NETWORK
TITLE =
//Blokada NA write
      A     "DB_HMI_Wozek".HMI_OUT.PB_Write_Kier_Rot;
      AN    "Bl_Na_Read_K_Rot";
      S     "Bl_Na_Write_K_Rot";
      A(;
      A     "Kier_Rot_Koniec_Send";
      FN    "Edge_M513.1";
      O     "Bl_Na_Read_K_Rot";
      O     "Help_M503.3";
      );
      R     "Bl_Na_Write_K_Rot";
      A     "Bl_Na_Write_K_Rot";
      =     #Aktywne_Write;
NETWORK
TITLE =
      O     "Bl_Na_Write_K_Rot";
      O     "Bl_Na_Read_K_Rot";
      =     #Aktywna_Funkcja;
